C01810=1212.912,107.053,-49.363,-178.523,5.760,148.578
C01811=1212.916,106.785,-49.342,-178.526,5.760,148.579
C01812=1212.922,106.536,-49.323,-178.528,5.758,148.579
C01813=1212.926,106.286,-49.305,-178.531,5.757,148.580
C01814=1212.931,106.037,-49.285,-178.533,5.756,148.581
C01815=1212.935,105.788,-49.266,-178.536,5.755,148.581
C01816=1212.941,105.539,-49.248,-178.539,5.754,148.582
C01817=1212.945,105.289,-49.229,-178.541,5.753,148.582
C01818=1212.950,105.040,-49.209,-178.544,5.752,148.583
C01819=1212.955,104.791,-49.191,-178.546,5.751,148.583
C01820=1212.960,104.542,-49.172,-178.549,5.750,148.584
C01821=1212.965,104.292,-49.154,-178.551,5.749,148.584
C01822=1212.969,104.043,-49.134,-178.554,5.748,148.585
C01823=1212.974,103.794,-49.115,-178.557,5.747,148.585
C01824=1212.979,103.544,-49.097,-178.559,5.746,148.586
C01825=1212.984,103.296,-49.078,-178.562,5.745,148.587
C01826=1212.989,103.046,-49.060,-178.564,5.744,148.587
C01827=1212.993,102.797,-49.040,-178.567,5.743,148.588
C01828=1212.998,102.548,-49.022,-178.570,5.742,148.588
C01829=1213.004,102.299,-49.003,-178.572,5.741,148.589
C01830=1213.008,102.049,-48.985,-178.574,5.740,148.589
C01831=1213.013,101.800,-48.965,-178.578,5.739,148.590
C01832=1213.018,101.550,-48.947,-178.580,5.738,148.590
C01833=1213.022,101.302,-48.928,-178.582,5.737,148.591
C01834=1213.028,101.052,-48.910,-178.585,5.737,148.592
C01835=1213.032,100.803,-48.891,-178.588,5.735,148.592
C01836=1213.037,100.554,-48.873,-178.590,5.734,148.593
C01837=1213.042,100.305,-48.853,-178.593,5.734,148.593
C01838=1213.046,100.055,-48.835,-178.596,5.732,148.594
C01839=1213.052,99.806,-48.816,-178.598,5.731,148.594
C01840=1213.057,99.557,-48.798,-178.600,5.730,148.595
C01841=1213.061,99.308,-48.779,-178.603,5.730,148.595
C01842=1213.066,99.058,-48.760,-178.606,5.728,148.596
C01843=1213.071,98.809,-48.742,-178.608,5.727,148.596
C01844=1213.075,98.560,-48.723,-178.611,5.727,148.597
C01845=1213.081,98.310,-48.704,-178.614,5.725,148.597
C01846=1213.086,98.061,-48.686,-178.616,5.724,148.598
C01847=1213.090,97.812,-48.667,-178.618,5.723,148.599
C01848=1213.095,97.563,-48.649,-178.621,5.723,148.599
C01849=1213.100,97.314,-48.630,-178.624,5.721,148.600
C01850=1213.104,97.064,-48.612,-178.626,5.721,148.600
C01851=1213.109,96.815,-48.594,-178.629,5.720,148.601
C01852=1213.115,96.565,-48.575,-178.632,5.719,148.602
C01853=1213.119,96.316,-48.556,-178.634,5.718,148.602
C01854=1213.124,96.067,-48.538,-178.637,5.717,148.603
C01855=1213.129,95.818,-48.520,-178.639,5.716,148.603
C01856=1213.134,95.569,-48.501,-178.642,5.715,148.604
C01857=1213.138,95.319,-48.483,-178.645,5.714,148.604
C01858=1213.143,95.070,-48.465,-178.647,5.713,148.605
C01859=1213.148,94.821,-48.447,-178.650,5.713,148.605
C01860=1213.154,94.572,-48.427,-178.652,5.711,148.606
C01861=1213.158,94.322,-48.409,-178.655,5.710,148.606
C01862=1213.163,94.073,-48.391,-178.658,5.710,148.607
C01863=1213.168,93.823,-48.373,-178.660,5.709,148.608
C01864=1213.172,93.575,-48.354,-178.663,5.707,148.608
C01865=1213.177,93.325,-48.335,-178.665,5.707,148.609
C01866=1213.182,93.076,-48.317,-178.668,5.706,148.609
C01867=1213.187,92.826,-48.299,-178.670,5.705,148.610
C01868=1213.192,92.577,-48.281,-178.673,5.703,148.610
C01869=1213.196,92.327,-48.263,-178.676,5.703,148.611
C01870=1213.201,92.079,-48.244,-178.678,5.702,148.612
C01871=1213.207,91.829,-48.226,-178.680,5.701,148.612
C01872=1213.212,91.580,-48.208,-178.683,5.700,148.613
C01873=1213.217,91.331,-48.190,-178.686,5.699,148.613
C01874=1213.221,91.081,-48.172,-178.688,5.698,148.614
C01875=1213.226,90.832,-48.154,-178.691,5.698,148.614
C01876=1213.231,90.583,-48.136,-178.694,5.696,148.615
C01877=1213.236,90.334,-48.118,-178.696,5.695,148.615
C01878=1213.241,90.084,-48.100,-178.699,5.695,148.616
C01879=1213.245,89.835,-48.080,-178.701,5.694,148.617
C01880=1213.250,89.586,-48.062,-178.704,5.693,148.617
C01881=1213.255,89.336,-48.044,-178.707,5.692,148.618
C01882=1213.260,89.087,-48.026,-178.709,5.691,148.618
C01883=1213.265,88.838,-48.008,-178.711,5.690,148.619
C01884=1213.270,88.589,-47.990,-178.714,5.690,148.620
C01885=1213.274,88.339,-47.972,-178.717,5.688,148.620
C01886=1213.279,88.090,-47.954,-178.719,5.687,148.621
C01887=1213.284,87.841,-47.936,-178.722,5.687,148.621
C01888=1213.289,87.591,-47.918,-178.724,5.686,148.622
C01889=1213.294,87.342,-47.900,-178.727,5.685,148.622
C01890=1213.299,87.093,-47.882,-178.730,5.684,148.623
C01891=1213.304,86.844,-47.864,-178.732,5.683,148.623
C01892=1213.308,86.594,-47.845,-178.735,5.682,148.624
C01893=1213.313,86.345,-47.828,-178.737,5.681,148.624
C01894=1213.318,86.095,-47.810,-178.740,5.680,148.625
C01895=1213.323,85.846,-47.792,-178.743,5.680,148.626
C01896=1213.328,85.597,-47.774,-178.745,5.679,148.626
C01897=1213.333,85.348,-47.756,-178.747,5.678,148.627
C01898=1213.338,85.098,-47.738,-178.750,5.677,148.628
C01899=1213.343,84.849,-47.720,-178.753,5.676,148.628
C01900=1213.348,84.600,-47.702,-178.755,5.675,148.629
C01901=1213.352,84.350,-47.684,-178.758,5.674,148.629
C01902=1213.357,84.101,-47.666,-178.760,5.674,148.630
C01903=1213.362,83.851,-47.649,-178.763,5.673,148.630
C01904=1213.367,83.602,-47.631,-178.766,5.672,148.631
C01905=1213.372,83.353,-47.613,-178.768,5.671,148.631
C01906=1213.377,83.104,-47.595,-178.771,5.670,148.632
C01907=1213.382,82.855,-47.577,-178.773,5.669,148.633
C01908=1213.387,82.605,-47.559,-178.776,5.669,148.633
C01909=1213.392,82.356,-47.542,-178.779,5.667,148.634
C01910=1213.397,82.106,-47.524,-178.781,5.667,148.634
C01911=1213.401,81.858,-47.506,-178.783,5.666,148.635
C01912=1213.406,81.589,-47.487,-178.786,5.665,148.636
C01913=1213.411,81.320,-47.468,-178.789,5.664,148.636
C01914=1213.416,81.052,-47.449,-178.792,5.663,148.637
C01915=1213.421,80.784,-47.429,-178.795,5.663,148.637
C01916=1213.427,80.534,-47.412,-178.798,5.661,148.638
C01917=1213.432,80.285,-47.394,-178.800,5.660,148.639
C01918=1213.436,80.036,-47.376,-178.803,5.660,148.639
C01919=1213.442,79.786,-47.359,-178.805,5.659,148.640
C01920=1213.447,79.537,-47.341,-178.807,5.658,148.640
C01921=1213.451,79.288,-47.323,-178.810,5.658,148.641
C01922=1213.456,79.038,-47.306,-178.813,5.656,148.642
C01923=1213.461,78.789,-47.288,-178.815,5.655,148.642
C01924=1213.466,78.540,-47.270,-178.818,5.655,148.643
C01925=1213.471,78.290,-47.253,-178.820,5.654,148.643
C01926=1213.476,78.041,-47.235,-178.823,5.653,148.644
C01927=1213.480,77.792,-47.218,-178.825,5.653,148.644
C01928=1213.485,77.542,-47.200,-178.828,5.651,148.645
C01929=1213.490,77.293,-47.182,-178.831,5.651,148.646
C01930=1213.495,77.044,-47.164,-178.833,5.650,148.646
C01931=1213.500,76.794,-47.148,-178.836,5.649,148.647
C01932=1213.505,76.545,-47.130,-178.838,5.649,148.647
C01933=1213.510,76.295,-47.112,-178.841,5.648,148.648
C01934=1213.515,76.046,-47.095,-178.844,5.646,148.649
C01935=1213.520,75.796,-47.077,-178.846,5.646,148.649
C01936=1213.524,75.547,-47.060,-178.849,5.645,148.650
C01937=1213.529,75.298,-47.042,-178.851,5.644,148.650
C01938=1213.534,75.048,-47.025,-178.854,5.644,148.651
C01939=1213.539,74.800,-47.008,-178.856,5.643,148.652
C01940=1213.544,74.551,-46.990,-178.859,5.642,148.652
C01941=1213.549,74.301,-46.972,-178.862,5.641,148.653
C01942=1213.554,74.052,-46.955,-178.864,5.640,148.653
C01943=1213.559,73.803,-46.938,-178.867,5.639,148.654
C01944=1213.564,73.553,-46.920,-178.869,5.639,148.654
C01945=1213.569,73.304,-46.902,-178.872,5.638,148.655
C01946=1213.573,73.054,-46.886,-178.874,5.637,148.656
C01947=1213.578,72.804,-46.869,-178.877,5.637,148.656
C01948=1213.583,72.555,-46.851,-178.880,5.635,148.657
C01949=1213.588,72.306,-46.834,-178.882,5.635,148.657
C01950=1213.593,72.057,-46.816,-178.885,5.634,148.658
C01951=1213.598,71.808,-46.799,-178.887,5.633,148.659
C01952=1213.603,71.559,-46.782,-178.890,5.633,148.659
C01953=1213.608,71.309,-46.764,-178.892,5.632,148.660
C01954=1213.613,71.059,-46.747,-178.895,5.631,148.660
C01955=1213.617,70.810,-46.730,-178.897,5.630,148.661
C01956=1213.622,70.560,-46.712,-178.900,5.629,148.662
C01957=1213.627,70.312,-46.695,-178.903,5.628,148.662
C01958=1213.632,70.062,-46.678,-178.905,5.628,148.663
C01959=1213.638,69.813,-46.661,-178.908,5.627,148.663
C01960=1213.642,69.564,-46.643,-178.910,5.626,148.664
C01961=1213.647,69.314,-46.626,-178.913,5.625,148.664
C01962=1213.652,69.065,-46.610,-178.915,5.625,148.665
C01963=1213.656,68.815,-46.592,-178.918,5.624,148.666
C01964=1213.662,68.566,-46.574,-178.921,5.623,148.666
C01965=1213.666,68.316,-46.558,-178.923,5.622,148.667
C01966=1213.672,68.067,-46.541,-178.926,5.621,148.668
C01967=1213.676,67.818,-46.523,-178.928,5.621,148.668
C01968=1213.681,67.568,-46.506,-178.931,5.620,148.669
C01969=1213.686,67.319,-46.489,-178.933,5.619,148.669
C01970=1213.691,67.070,-46.471,-178.936,5.619,148.670
C01971=1213.696,66.821,-46.455,-178.938,5.618,148.671
C01972=1213.701,66.571,-46.438,-178.941,5.617,148.671
C01973=1213.706,66.322,-46.421,-178.944,5.616,148.672
C01974=1213.711,66.072,-46.404,-178.946,5.615,148.672
C01975=1213.715,65.823,-46.387,-178.949,5.615,148.673
C01976=1213.720,65.573,-46.369,-178.951,5.614,148.673
C01977=1213.725,65.324,-46.353,-178.954,5.613,148.674
C01978=1213.730,65.075,-46.336,-178.956,5.613,148.675
C01979=1213.735,64.825,-46.319,-178.959,5.612,148.675
C01980=1213.740,64.576,-46.301,-178.961,5.611,148.676
C01981=1213.745,64.327,-46.285,-178.964,5.611,148.677
C01982=1213.750,64.077,-46.268,-178.966,5.610,148.677
C01983=1213.755,63.828,-46.251,-178.970,5.609,148.678
C01984=1213.760,63.578,-46.234,-178.972,5.608,148.678
C01985=1213.764,63.329,-46.217,-178.974,5.607,148.679
C01986=1213.770,63.079,-46.200,-178.977,5.607,148.680
C01987=1213.774,62.831,-46.183,-178.980,5.606,148.680
C01988=1213.779,62.581,-46.166,-178.982,5.605,148.681
C01989=1213.785,62.332,-46.149,-178.985,5.605,148.681
C01990=1213.789,62.083,-46.132,-178.987,5.604,148.682
C01991=1213.794,61.833,-46.115,-178.990,5.604,148.683
C01992=1213.799,61.583,-46.098,-178.992,5.603,148.683
C01993=1213.804,61.334,-46.082,-178.995,5.602,148.684
C01994=1213.809,61.085,-46.065,-178.997,5.602,148.685
C01995=1213.814,60.835,-46.048,-179.000,5.600,148.685
C01996=1213.819,60.585,-46.031,-179.003,5.599,148.686
C01997=1213.824,60.337,-46.015,-179.005,5.599,148.686
C01998=1213.828,60.087,-45.998,-179.008,5.598,148.687
C01999=1213.834,59.837,-45.981,-179.010,5.598,148.688
C02000=1213.839,59.589,-45.964,-179.013,5.597,148.688
C02001=1213.843,59.339,-45.948,-179.015,5.596,148.689
C02002=1213.848,59.089,-45.930,-179.018,5.596,148.689
C02003=1213.853,58.840,-45.914,-179.020,5.595,148.690
C02004=1213.858,58.591,-45.898,-179.023,5.594,148.691
C02005=1213.863,58.341,-45.880,-179.025,5.594,148.691
C02006=1213.868,58.092,-45.864,-179.028,5.593,148.692
C02007=1213.873,57.843,-45.847,-179.031,5.592,148.692
C02008=1213.878,57.593,-45.830,-179.033,5.592,148.693
C02009=1213.882,57.344,-45.813,-179.035,5.591,148.694
C02010=1213.887,57.095,-45.797,-179.039,5.590,148.694
C02011=1213.893,56.844,-45.780,-179.041,5.589,148.695
C02012=1213.898,56.596,-45.764,-179.044,5.588,148.696
C02013=1213.903,56.346,-45.748,-179.046,5.588,148.696
C02014=1213.907,56.097,-45.731,-179.049,5.587,148.697
C02015=1213.913,55.848,-45.714,-179.051,5.586,148.697
C02016=1213.918,55.579,-45.696,-179.054,5.586,148.698
C02017=1213.923,55.311,-45.679,-179.056,5.585,148.699
C02018=1213.928,55.042,-45.660,-179.059,5.585,148.699
C02019=1213.934,54.774,-45.642,-179.062,5.583,148.700
C02020=1213.938,54.524,-45.626,-179.065,5.583,148.701
C02021=1213.944,54.275,-45.610,-179.068,5.582,148.701
C02022=1213.949,54.025,-45.593,-179.070,5.581,148.702
C02023=1213.953,53.776,-45.576,-179.072,5.581,148.702
C02024=1213.958,53.527,-45.560,-179.075,5.580,148.703
C02025=1213.963,53.277,-45.544,-179.078,5.580,148.704
C02026=1213.968,53.028,-45.528,-179.080,5.579,148.704
C02027=1213.973,52.778,-45.510,-179.082,5.578,148.705
C02028=1213.978,52.529,-45.494,-179.085,5.578,148.706
C02029=1213.983,52.279,-45.478,-179.088,5.577,148.706
C02030=1213.988,52.030,-45.461,-179.090,5.577,148.707
C02031=1213.993,51.781,-45.445,-179.092,5.576,148.707
C02032=1213.997,51.532,-45.428,-179.095,5.575,148.708
C02033=1214.003,51.282,-45.412,-179.098,5.575,148.709
C02034=1214.008,51.032,-45.396,-179.100,5.574,148.709
C02035=1214.012,50.783,-45.379,-179.103,5.573,148.710
C02036=1214.018,50.533,-45.363,-179.105,5.573,148.710
C02037=1214.022,50.284,-45.347,-179.108,5.572,148.711
C02038=1214.027,50.035,-45.330,-179.110,5.571,148.712
C02039=1214.032,49.785,-45.314,-179.113,5.571,148.712
C02040=1214.037,49.536,-45.298,-179.116,5.570,148.713
C02041=1214.042,49.287,-45.281,-179.118,5.569,148.714
C02042=1214.048,49.037,-45.265,-179.120,5.569,148.714
C02043=1214.052,48.788,-45.249,-179.123,5.568,148.715
C02044=1214.057,48.538,-45.233,-179.126,5.568,148.716
C02045=1214.062,48.289,-45.216,-179.128,5.567,148.716
C02046=1214.067,48.039,-45.200,-179.131,5.566,148.717
C02047=1214.072,47.790,-45.184,-179.133,5.566,148.717
C02048=1214.077,47.540,-45.167,-179.136,5.565,148.718
C02049=1214.082,47.291,-45.152,-179.138,5.565,148.719
C02050=1214.086,47.042,-45.135,-179.141,5.564,148.719
C02051=1214.092,46.792,-45.120,-179.144,5.564,148.720
C02052=1214.096,46.543,-45.103,-179.146,5.563,148.720
C02053=1214.101,46.294,-45.087,-179.149,5.562,148.721
C02054=1214.106,46.044,-45.071,-179.151,5.562,148.722
C02055=1214.111,45.795,-45.054,-179.154,5.561,148.723
C02056=1214.116,45.545,-45.038,-179.156,5.560,148.723
C02057=1214.121,45.296,-45.022,-179.159,5.560,148.724
C02058=1214.126,45.046,-45.006,-179.161,5.559,148.724
C02059=1214.131,44.797,-44.990,-179.164,5.558,148.725
C02060=1214.136,44.548,-44.974,-179.167,5.558,148.726
C02061=1214.141,44.298,-44.958,-179.169,5.557,148.726
C02062=1214.146,44.049,-44.942,-179.171,5.556,148.727
C02063=1214.151,43.799,-44.926,-179.174,5.556,148.727
C02064=1214.156,43.550,-44.910,-179.177,5.555,148.728
C02065=1214.161,43.300,-44.894,-179.179,5.555,148.729
C02066=1214.166,43.051,-44.878,-179.182,5.554,148.729
C02067=1214.171,42.801,-44.862,-179.184,5.554,148.730
C02068=1214.176,42.552,-44.845,-179.187,5.553,148.731
C02069=1214.181,42.303,-44.830,-179.189,5.552,148.731
C02070=1214.186,42.053,-44.814,-179.192,5.552,148.732
C02071=1214.191,41.804,-44.797,-179.195,5.551,148.733
C02072=1214.196,41.554,-44.781,-179.197,5.551,148.733
C02073=1214.201,41.304,-44.766,-179.200,5.550,148.734
C02074=1214.206,41.055,-44.749,-179.202,5.549,148.734
C02075=1214.211,40.806,-44.734,-179.205,5.549,148.735
C02076=1214.216,40.557,-44.717,-179.207,5.548,148.736
C02077=1214.220,40.307,-44.702,-179.210,5.548,148.736
C02078=1214.226,40.058,-44.686,-179.213,5.547,148.737
C02079=1214.230,39.807,-44.670,-179.215,5.546,148.738
C02080=1214.235,39.559,-44.654,-179.217,5.546,148.738
C02081=1214.241,39.309,-44.639,-179.220,5.545,148.739
C02082=1214.246,39.059,-44.623,-179.223,5.544,148.740
C02083=1214.251,38.810,-44.606,-179.225,5.544,148.740
C02084=1214.256,38.561,-44.591,-179.228,5.543,148.741
C02085=1214.260,38.311,-44.575,-179.231,5.543,148.742
C02086=1214.266,38.062,-44.560,-179.233,5.542,148.742
C02087=1214.270,37.812,-44.543,-179.235,5.541,148.743
C02088=1214.275,37.563,-44.527,-179.238,5.541,148.743
C02089=1214.281,37.314,-44.512,-179.241,5.540,148.744
C02090=1214.286,37.063,-44.496,-179.243,5.540,148.745
C02091=1214.290,36.815,-44.480,-179.246,5.539,148.745
C02092=1214.295,36.566,-44.465,-179.248,5.538,148.746
C02093=1214.300,36.315,-44.449,-179.251,5.538,148.746
C02094=1214.306,36.066,-44.433,-179.253,5.537,148.747
C02095=1214.311,35.817,-44.417,-179.256,5.537,148.748
C02096=1214.315,35.567,-44.401,-179.258,5.537,148.749
C02097=1214.320,35.318,-44.386,-179.261,5.536,148.749
C02098=1214.325,35.069,-44.370,-179.263,5.536,148.750
C02099=1214.330,34.819,-44.354,-179.265,5.535,148.750
C02100=1214.335,34.569,-44.339,-179.268,5.534,148.751
C02101=1214.340,34.320,-44.324,-179.271,5.534,148.752
C02102=1214.346,34.071,-44.308,-179.273,5.533,148.752
C02103=1214.350,33.821,-44.291,-179.276,5.533,148.753
C02104=1214.355,33.572,-44.276,-179.279,5.532,148.754
C02105=1214.360,33.323,-44.261,-179.281,5.531,148.754
C02106=1214.365,33.073,-44.245,-179.283,5.531,148.755
C02107=1214.370,32.823,-44.229,-179.286,5.530,148.755
C02108=1214.375,32.574,-44.214,-179.289,5.530,148.756
C02109=1214.380,32.324,-44.198,-179.291,5.529,148.757
C02110=1214.385,32.075,-44.183,-179.294,5.529,148.758
C02111=1214.390,31.825,-44.168,-179.297,5.528,148.758
C02112=1214.395,31.576,-44.152,-179.299,5.527,148.759
C02113=1214.400,31.326,-44.136,-179.301,5.528,148.759
C02114=1214.405,31.077,-44.121,-179.304,5.527,148.760
C02115=1214.410,30.827,-44.106,-179.306,5.527,148.761
C02116=1214.415,30.578,-44.090,-179.309,5.526,148.761
C02117=1214.419,30.328,-44.075,-179.312,5.525,148.762
C02118=1214.425,30.079,-44.059,-179.314,5.525,148.763
C02119=1214.430,29.829,-44.044,-179.316,5.524,148.763
C02120=1214.435,29.561,-44.027,-179.319,5.523,148.764
C02121=1214.441,29.293,-44.010,-179.322,5.523,148.765
C02122=1214.446,29.024,-43.994,-179.325,5.523,148.765
C02123=1214.451,28.755,-43.977,-179.327,5.522,148.766
C02124=1214.456,28.505,-43.961,-179.330,5.522,148.767
C02125=1214.461,28.256,-43.946,-179.332,5.521,148.767
C02126=1214.466,28.007,-43.931,-179.335,5.520,148.768
C02127=1214.471,27.758,-43.915,-179.337,5.520,148.769
C02128=1214.477,27.507,-43.900,-179.340,5.519,148.769
C02129=1214.481,27.258,-43.885,-179.343,5.519,148.770
C02130=1214.487,27.008,-43.869,-179.345,5.518,148.771
C02131=1214.491,26.759,-43.854,-179.348,5.518,148.771
C02132=1214.497,26.510,-43.839,-179.350,5.517,148.772
C02133=1214.501,26.260,-43.824,-179.352,5.517,148.772
C02134=1214.506,26.011,-43.808,-179.355,5.516,148.773
C02135=1214.511,25.761,-43.792,-179.358,5.516,148.774
C02136=1214.516,25.512,-43.778,-179.360,5.515,148.774
C02137=1214.522,25.262,-43.762,-179.363,5.515,148.775
C02138=1214.526,25.013,-43.747,-179.365,5.514,148.776
C02139=1214.531,24.763,-43.732,-179.368,5.514,148.777
C02140=1214.536,24.514,-43.717,-179.370,5.513,148.777
C02141=1214.541,24.264,-43.701,-179.373,5.512,148.778
C02142=1214.546,24.015,-43.687,-179.376,5.512,148.778
C02143=1214.552,23.765,-43.671,-179.378,5.511,148.779
C02144=1214.556,23.516,-43.656,-179.380,5.512,148.780
C02145=1214.561,23.266,-43.640,-179.383,5.511,148.780
C02146=1214.566,23.016,-43.626,-179.386,5.511,148.781
C02147=1214.571,22.767,-43.610,-179.388,5.510,148.782
C02148=1214.576,22.518,-43.595,-179.390,5.509,148.782
C02149=1214.581,22.269,-43.580,-179.393,5.509,148.783
C02150=1214.586,22.019,-43.565,-179.396,5.508,148.784
C02151=1214.592,21.769,-43.550,-179.398,5.508,148.784
C02152=1214.596,21.520,-43.535,-179.401,5.507,148.785
C02153=1214.601,21.270,-43.519,-179.403,5.507,148.786
C02154=1214.606,21.021,-43.505,-179.406,5.507,148.786
C02155=1214.611,20.771,-43.490,-179.408,5.506,148.787
C02156=1214.616,20.522,-43.474,-179.411,5.506,148.788
C02157=1214.621,20.272,-43.460,-179.413,5.505,148.788
C02158=1214.627,20.023,-43.444,-179.416,5.504,148.789
C02159=1214.631,19.774,-43.429,-179.418,5.504,148.789
C02160=1214.637,19.524,-43.414,-179.421,5.503,148.790
C02161=1214.642,19.275,-43.399,-179.423,5.504,148.791
C02162=1214.646,19.025,-43.385,-179.426,5.503,148.791
C02163=1214.652,18.776,-43.369,-179.428,5.503,148.792
C02164=1214.656,18.527,-43.354,-179.431,5.502,148.793
C02165=1214.661,18.276,-43.340,-179.433,5.501,148.793
C02166=1214.666,18.027,-43.324,-179.436,5.501,148.794
C02167=1214.671,17.778,-43.309,-179.439,5.500,148.795
C02168=1214.677,17.528,-43.294,-179.441,5.500,148.795
C02169=1214.681,17.278,-43.279,-179.443,5.500,148.796
C02170=1214.686,17.029,-43.265,-179.446,5.499,148.797
C02171=1214.692,16.779,-43.249,-179.449,5.499,148.797
C02172=1214.697,16.530,-43.235,-179.451,5.498,148.798
C02173=1214.701,16.281,-43.220,-179.454,5.498,148.799
C02174=1214.707,16.031,-43.205,-179.456,5.497,148.799
C02175=1214.712,15.781,-43.190,-179.459,5.496,148.800
C02176=1214.716,15.532,-43.176,-179.461,5.496,148.801
C02177=1214.722,15.282,-43.160,-179.463,5.496,148.801
C02178=1214.727,15.033,-43.146,-179.466,5.496,148.802
C02179=1214.731,14.784,-43.131,-179.469,5.495,148.803
C02180=1214.737,14.534,-43.116,-179.471,5.494,148.803
C02181=1214.742,14.284,-43.101,-179.474,5.494,148.804
C02182=1214.747,14.035,-43.087,-179.477,5.493,148.805
C02183=1214.751,13.786,-43.072,-179.479,5.493,148.805
C02184=1214.757,13.536,-43.057,-179.481,5.493,148.806
C02185=1214.762,13.287,-43.042,-179.484,5.492,148.807
C02186=1214.767,13.037,-43.028,-179.486,5.492,148.807
C02187=1214.771,12.788,-43.013,-179.489,5.491,148.808
C02188=1214.777,12.538,-42.998,-179.491,5.491,148.809
C02189=1214.782,12.288,-42.984,-179.494,5.490,148.809
C02190=1214.787,12.039,-42.969,-179.496,5.491,148.810
C02191=1214.792,11.789,-42.955,-179.499,5.490,148.811
C02192=1214.797,11.540,-42.939,-179.501,5.490,148.811
C02193=1214.802,11.290,-42.925,-179.504,5.489,148.812
C02194=1214.807,11.040,-42.910,-179.506,5.488,148.812
C02195=1214.812,10.791,-42.895,-179.509,5.488,148.813
C02196=1214.817,10.541,-42.881,-179.512,5.487,148.814
C02197=1214.822,10.292,-42.866,-179.514,5.487,148.814
C02198=1214.827,10.042,-42.851,-179.516,5.487,148.815
C02199=1214.832,9.793,-42.837,-179.519,5.486,148.816
C02200=1214.837,9.543,-42.823,-179.522,5.486,148.817
C02201=1214.842,9.295,-42.808,-179.524,5.485,148.817
C02202=1214.848,9.045,-42.793,-179.527,5.485,148.818
C02203=1214.853,8.795,-42.779,-179.529,5.485,148.819
C02204=1214.857,8.546,-42.764,-179.531,5.484,148.819
C02205=1214.862,8.296,-42.750,-179.534,5.484,148.820
C02206=1214.867,8.046,-42.735,-179.536,5.483,148.820
C02207=1214.872,7.797,-42.721,-179.539,5.483,148.821
C02208=1214.878,7.547,-42.706,-179.542,5.482,148.822
C02209=1214.883,7.298,-42.691,-179.544,5.482,148.822
C02210=1214.887,7.048,-42.677,-179.546,5.482,148.823
C02211=1214.892,6.798,-42.663,-179.549,5.481,148.824
C02212=1214.897,6.549,-42.648,-179.552,5.481,148.825
C02213=1214.903,6.300,-42.634,-179.554,5.480,148.825
C02214=1214.908,6.050,-42.619,-179.557,5.480,148.826
C02215=1214.913,5.801,-42.605,-179.559,5.480,148.826
C02216=1214.917,5.552,-42.590,-179.561,5.479,148.827
C02217=1214.923,5.302,-42.575,-179.564,5.479,148.828
C02218=1214.928,5.052,-42.561,-179.567,5.478,148.828
C02219=1214.933,4.802,-42.547,-179.569,5.478,148.829
C02220=1214.938,4.552,-42.533,-179.571,5.478,148.830
C02221=1214.943,4.303,-42.519,-179.574,5.478,148.831
C02222=1214.948,4.054,-42.504,-179.577,5.477,148.831
C02223=1214.953,3.805,-42.489,-179.579,5.476,148.832
C02224=1214.958,3.535,-42.474,-179.582,5.476,148.833
C02225=1214.963,3.266,-42.459,-179.585,5.475,148.833
C02226=1214.969,2.998,-42.443,-179.587,5.475,148.834
C02227=1214.975,2.728,-42.427,-179.590,5.474,148.835
C02228=1214.980,2.479,-42.413,-179.592,5.475,148.835
C02229=1214.985,2.229,-42.399,-179.595,5.474,148.836
C02230=1214.990,1.979,-42.385,-179.597,5.474,148.837
C02231=1214.995,1.730,-42.371,-179.600,5.473,148.837
C02232=1215.000,1.480,-42.356,-179.603,5.473,148.838
C02233=1215.005,1.231,-42.341,-179.605,5.473,148.839
C02234=1215.010,0.982,-42.327,-179.607,5.472,148.839
C02235=1215.015,0.732,-42.313,-179.610,5.472,148.840
C02236=1215.020,0.482,-42.299,-179.613,5.471,148.841
C02237=1215.025,0.233,-42.285,-179.615,5.471,148.842
C02238=1215.030,-0.017,-42.270,-179.617,5.471,148.842
C02239=1215.035,-0.266,-42.257,-179.620,5.470,148.843
C02240=1215.040,-0.515,-42.243,-179.622,5.470,148.843
C02241=1215.045,-0.765,-42.228,-179.625,5.469,148.844
C02242=1215.050,-1.015,-42.214,-179.627,5.469,148.845
C02243=1215.055,-1.264,-42.200,-179.630,5.469,148.845
C02244=1215.060,-1.513,-42.186,-179.632,5.469,148.846
C02245=1215.065,-1.763,-42.172,-179.635,5.468,148.847
C02246=1215.070,-2.013,-42.157,-179.638,5.468,148.847
C02247=1215.075,-2.263,-42.143,-179.640,5.467,148.848
C02248=1215.081,-2.512,-42.129,-179.642,5.467,148.849
C02249=1215.086,-2.762,-42.116,-179.645,5.467,148.850
C02250=1215.091,-3.012,-42.101,-179.648,5.466,148.850
C02251=1215.096,-3.261,-42.087,-179.650,5.466,148.851
C02252=1215.101,-3.510,-42.073,-179.652,5.465,148.851
C02253=1215.106,-3.760,-42.060,-179.654,5.465,148.852
C02254=1215.111,-4.010,-42.045,-179.657,5.465,148.853
C02255=1215.116,-4.259,-42.031,-179.660,5.464,148.853
C02256=1215.121,-4.508,-42.017,-179.662,5.464,148.854
C02257=1215.126,-4.758,-42.003,-179.664,5.464,148.855
C02258=1215.131,-5.008,-41.989,-179.667,5.464,148.856
C02259=1215.137,-5.257,-41.975,-179.670,5.463,148.856
C02260=1215.141,-5.507,-41.962,-179.672,5.463,148.857
C02261=1215.146,-5.756,-41.947,-179.675,5.462,148.858
C02262=1215.151,-6.006,-41.933,-179.677,5.462,148.858
C02263=1215.157,-6.255,-41.919,-179.680,5.462,148.859
C02264=1215.162,-6.505,-41.905,-179.682,5.461,148.860
C02265=1215.167,-6.755,-41.891,-179.685,5.461,148.860
C02266=1215.172,-7.004,-41.878,-179.687,5.461,148.861
C02267=1215.177,-7.254,-41.864,-179.689,5.460,148.862
C02268=1215.182,-7.503,-41.849,-179.692,5.460,148.862
C02269=1215.187,-7.752,-41.836,-179.695,5.459,148.863
C02270=1215.192,-8.003,-41.822,-179.697,5.460,148.864
C02271=1215.197,-8.252,-41.808,-179.699,5.459,148.864
C02272=1215.202,-8.501,-41.794,-179.702,5.459,148.865
C02273=1215.207,-8.751,-41.780,-179.705,5.458,148.866
C02274=1215.212,-9.001,-41.767,-179.707,5.458,148.866
C02275=1215.217,-9.250,-41.753,-179.709,5.458,148.867
C02276=1215.222,-9.499,-41.739,-179.712,5.457,148.868
C02277=1215.227,-9.750,-41.725,-179.715,5.457,148.868
C02278=1215.233,-9.999,-41.711,-179.717,5.456,148.869
C02279=1215.237,-10.248,-41.698,-179.720,5.457,148.870
C02280=1215.242,-10.498,-41.684,-179.722,5.456,148.870
C02281=1215.248,-10.748,-41.670,-179.724,5.455,148.871
C02282=1215.253,-10.997,-41.656,-179.727,5.455,148.872
C02283=1215.257,-11.247,-41.642,-179.729,5.455,148.872
C02284=1215.263,-11.496,-41.629,-179.732,5.455,148.873
C02285=1215.268,-11.746,-41.615,-179.734,5.454,148.874
C02286=1215.272,-11.995,-41.601,-179.737,5.454,148.874
C02287=1215.278,-12.245,-41.588,-179.739,5.454,148.875
C02288=1215.283,-12.495,-41.574,-179.742,5.453,148.876
C02289=1215.289,-12.744,-41.561,-179.744,5.453,148.877
C02290=1215.293,-12.994,-41.547,-179.747,5.452,148.877
C02291=1215.298,-13.243,-41.533,-179.749,5.453,148.878
C02292=1215.304,-13.493,-41.519,-179.752,5.452,148.879
C02293=1215.308,-13.742,-41.506,-179.754,5.452,148.879
C02294=1215.314,-13.992,-41.493,-179.757,5.451,148.880
C02295=1215.319,-14.242,-41.478,-179.759,5.451,148.880
C02296=1215.323,-14.491,-41.465,-179.761,5.451,148.881
C02297=1215.329,-14.741,-41.451,-179.764,5.450,148.882
C02298=1215.333,-14.990,-41.438,-179.767,5.450,148.883
C02299=1215.339,-15.240,-41.424,-179.769,5.450,148.883
C02300=1215.344,-15.490,-41.410,-179.771,5.450,148.884
C02301=1215.349,-15.739,-41.398,-179.774,5.449,148.885
C02302=1215.354,-15.989,-41.383,-179.776,5.449,148.885
C02303=1215.359,-16.239,-41.370,-179.779,5.449,148.886
C02304=1215.364,-16.488,-41.356,-179.781,5.448,148.887
C02305=1215.369,-16.738,-41.343,-179.784,5.448,148.887
C02306=1215.374,-16.987,-41.330,-179.786,5.448,148.888
C02307=1215.380,-17.237,-41.316,-179.789,5.448,148.889
C02308=1215.385,-17.486,-41.302,-179.792,5.447,148.889
C02309=1215.390,-17.736,-41.289,-179.794,5.447,148.890
C02310=1215.395,-17.985,-41.275,-179.796,5.447,148.891
C02311=1215.400,-18.235,-41.262,-179.798,5.446,148.891
C02312=1215.405,-18.484,-41.248,-179.801,5.446,148.892
C02313=1215.410,-18.734,-41.235,-179.804,5.445,148.893
C02314=1215.415,-18.983,-41.221,-179.806,5.446,148.893
C02315=1215.421,-19.233,-41.208,-179.808,5.445,148.894
C02316=1215.426,-19.483,-41.195,-179.811,5.445,148.895
C02317=1215.431,-19.732,-41.181,-179.813,5.445,148.895
C02318=1215.436,-19.982,-41.168,-179.816,5.444,148.896
C02319=1215.441,-20.231,-41.154,-179.819,5.444,148.897
C02320=1215.446,-20.481,-41.142,-179.821,5.443,148.898
C02321=1215.451,-20.731,-41.128,-179.823,5.444,148.898
C02322=1215.456,-20.980,-41.115,-179.826,5.443,148.899
C02323=1215.461,-21.230,-41.101,-179.829,5.443,148.900
C02324=1215.466,-21.479,-41.089,-179.831,5.443,148.900
C02325=1215.471,-21.729,-41.074,-179.833,5.443,148.901
C02326=1215.476,-21.979,-41.062,-179.836,5.442,148.902
C02327=1215.482,-22.229,-41.048,-179.839,5.442,148.902
C02328=1215.486,-22.498,-41.034,-179.841,5.442,148.903
C02329=1215.492,-22.767,-41.019,-179.843,5.441,148.904
C02330=1215.498,-23.037,-41.005,-179.846,5.441,148.905
C02331=1215.503,-23.306,-40.990,-179.849,5.440,148.905
C02332=1215.509,-23.555,-40.977,-179.851,5.440,148.906
C02333=1215.513,-23.805,-40.964,-179.853,5.440,148.907
C02334=1215.519,-24.055,-40.951,-179.856,5.440,148.907
C02335=1215.523,-24.304,-40.937,-179.859,5.439,148.908
C02336=1215.529,-24.554,-40.924,-179.861,5.440,148.909
C02337=1215.534,-24.803,-40.912,-179.864,5.439,148.909
C02338=1215.539,-25.053,-40.899,-179.866,5.439,148.910
C02339=1215.544,-25.302,-40.885,-179.869,5.438,148.911
C02340=1215.549,-25.552,-40.872,-179.871,5.438,148.911
C02341=1215.555,-25.802,-40.858,-179.874,5.438,148.912
C02342=1215.559,-26.052,-40.846,-179.876,5.437,148.913
C02343=1215.564,-26.301,-40.832,-179.878,5.438,148.914
C02344=1215.570,-26.550,-40.819,-179.880,5.437,148.914
C02345=1215.574,-26.800,-40.806,-179.883,5.436,148.915
C02346=1215.580,-27.050,-40.793,-179.885,5.437,148.915
C02347=1215.585,-27.300,-40.780,-179.888,5.436,148.916
C02348=1215.590,-27.549,-40.767,-179.891,5.436,148.917
C02349=1215.596,-27.798,-40.753,-179.893,5.435,148.918
C02350=1215.600,-28.048,-40.740,-179.895,5.436,148.918
C02351=1215.605,-28.298,-40.728,-179.898,5.435,148.919
C02352=1215.610,-28.548,-40.714,-179.901,5.435,148.920
C02353=1215.616,-28.797,-40.702,-179.903,5.435,148.920
C02354=1215.621,-29.047,-40.689,-179.905,5.434,148.921
C02355=1215.626,-29.297,-40.675,-179.908,5.434,148.922
C02356=1215.631,-29.546,-40.662,-179.910,5.434,148.922
C02357=1215.636,-29.795,-40.650,-179.913,5.434,148.923
C02358=1215.641,-30.045,-40.636,-179.915,5.433,148.924
C02359=1215.646,-30.295,-40.623,-179.918,5.434,148.925
C02360=1215.651,-30.545,-40.610,-179.920,5.433,148.925
C02361=1215.657,-30.794,-40.597,-179.923,5.433,148.926
C02362=1215.662,-31.044,-40.585,-179.924,5.433,148.926
C02363=1215.666,-31.294,-40.572,-179.927,5.432,148.927
C02364=1215.671,-31.543,-40.559,-179.930,5.432,148.928
C02365=1215.677,-31.793,-40.546,-179.932,5.431,148.928
C02366=1215.682,-32.043,-40.533,-179.934,5.432,148.929
C02367=1215.687,-32.292,-40.520,-179.937,5.431,148.930
C02368=1215.692,-32.541,-40.508,-179.940,5.431,148.931
C02369=1215.697,-32.792,-40.494,-179.942,5.431,148.931
C02370=1215.702,-33.041,-40.482,-179.945,5.430,148.932
C02371=1215.708,-33.290,-40.469,-179.947,5.430,148.933
C02372=1215.712,-33.540,-40.456,-179.949,5.430,148.933
C02373=1215.718,-33.790,-40.443,-179.952,5.430,148.934
C02374=1215.723,-34.039,-40.430,-179.955,5.429,148.935
C02375=1215.728,-34.289,-40.418,-179.957,5.430,148.935
C02376=1215.733,-34.539,-40.405,-179.959,5.429,148.936
C02377=1215.739,-34.788,-40.391,-179.962,5.429,148.937
C02378=1215.744,-35.038,-40.379,-179.964,5.429,148.938
C02379=1215.748,-35.288,-40.366,-179.967,5.429,148.938
C02380=1215.753,-35.537,-40.353,-179.969,5.428,148.939
C02381=1215.759,-35.786,-40.341,-179.971,5.428,148.939
C02382=1215.764,-36.036,-40.327,-179.974,5.427,148.940
C02383=1215.769,-36.286,-40.314,-179.976,5.427,148.941
C02384=1215.774,-36.535,-40.302,-179.978,5.427,148.942
C02385=1215.779,-36.784,-40.289,-179.981,5.427,148.942
C02386=1215.784,-37.035,-40.277,-179.984,5.426,148.943
C02387=1215.790,-37.285,-40.264,-179.986,5.427,148.944
C02388=1215.795,-37.534,-40.251,-179.988,5.426,148.944
C02389=1215.800,-37.783,-40.239,-179.991,5.426,148.945
C02390=1215.805,-38.033,-40.226,-179.993,5.426,148.946
C02391=1215.810,-38.283,-40.213,-179.996,5.426,148.946
C02392=1215.815,-38.532,-40.200,-179.999,5.425,148.947
C02393=1215.820,-38.782,-40.189,179.999,5.425,148.948
C02394=1215.826,-39.032,-40.175,179.997,5.425,148.949
C02395=1215.831,-39.282,-40.162,179.994,5.425,148.949
C02396=1215.836,-39.531,-40.150,179.992,5.425,148.950
C02397=1215.841,-39.780,-40.137,179.989,5.424,148.951
C02398=1215.846,-40.030,-40.125,179.988,5.424,148.951
C02399=1215.851,-40.280,-40.112,179.985,5.424,148.952
C02400=1215.856,-40.530,-40.100,179.982,5.423,148.952
C02401=1215.861,-40.779,-40.087,179.980,5.424,148.953
C02402=1215.866,-41.028,-40.075,179.978,5.423,148.954
C02403=1215.872,-41.278,-40.063,179.975,5.423,148.955
C02404=1215.876,-41.528,-40.050,179.973,5.423,148.955
C02405=1215.882,-41.778,-40.037,179.970,5.423,148.956
C02406=1215.887,-42.027,-40.024,179.968,5.422,148.957
C02407=1215.893,-42.277,-40.012,179.965,5.422,148.957
C02408=1215.898,-42.526,-39.999,179.963,5.422,148.958
C02409=1215.902,-42.776,-39.986,179.960,5.422,148.959
C02410=1215.907,-43.026,-39.974,179.958,5.422,148.960
C02411=1215.913,-43.276,-39.962,179.955,5.421,148.960
C02412=1215.918,-43.525,-39.949,179.953,5.421,148.961
C02413=1215.923,-43.774,-39.937,179.951,5.421,148.962
C02414=1215.928,-44.025,-39.925,179.948,5.421,148.962
C02415=1215.933,-44.274,-39.912,179.946,5.421,148.963
C02416=1215.938,-44.523,-39.899,179.944,5.420,148.963
C02417=1215.944,-44.773,-39.887,179.941,5.420,148.964
C02418=1215.949,-45.023,-39.875,179.939,5.420,148.965
C02419=1215.954,-45.272,-39.862,179.936,5.420,148.966
C02420=1215.959,-45.522,-39.850,179.934,5.419,148.966
C02421=1215.964,-45.772,-39.837,179.932,5.420,148.967
C02422=1215.969,-46.021,-39.825,179.929,5.419,148.968
C02423=1215.974,-46.271,-39.813,179.926,5.419,148.968
C02424=1215.979,-46.521,-39.800,179.924,5.419,148.969
C02425=1215.985,-46.771,-39.788,179.921,5.418,148.970
C02426=1215.990,-47.020,-39.776,179.919,5.419,148.971
C02427=1215.995,-47.269,-39.763,179.917,5.418,148.971
C02428=1216.001,-47.519,-39.751,179.914,5.418,148.972
C02429=1216.005,-47.769,-39.738,179.912,5.418,148.973
C02430=1216.010,-48.019,-39.727,179.909,5.418,148.973
C02431=1216.015,-48.268,-39.714,179.907,5.417,148.974
C02432=1216.022,-48.538,-39.701,179.905,5.418,148.975
C02433=1216.027,-48.808,-39.688,179.902,5.417,148.975
C02434=1216.032,-49.078,-39.675,179.899,5.417,148.976
C02435=1216.038,-49.348,-39.662,179.897,5.416,148.977
C02436=1216.043,-49.597,-39.649,179.894,5.416,148.978
C02437=1216.048,-49.848,-39.637,179.892,5.416,148.978
C02438=1216.053,-50.097,-39.625,179.890,5.416,148.979
C02439=1216.058,-50.347,-39.613,179.887,5.416,148.980
C02440=1216.063,-50.596,-39.600,179.884,5.415,148.980
C02441=1216.069,-50.846,-39.588,179.882,5.416,148.981
C02442=1216.073,-51.095,-39.576,179.880,5.415,148.982
C02443=1216.079,-51.345,-39.564,179.877,5.415,148.982
C02444=1216.084,-51.594,-39.552,179.875,5.415,148.983
C02445=1216.089,-51.844,-39.540,179.872,5.415,148.984
C02446=1216.094,-52.094,-39.527,179.870,5.415,148.985
C02447=1216.100,-52.344,-39.515,179.868,5.414,148.985
C02448=1216.105,-52.593,-39.503,179.865,5.414,148.986
C02449=1216.110,-52.843,-39.491,179.863,5.414,148.986
C02450=1216.115,-53.093,-39.480,179.861,5.414,148.987
C02451=1216.120,-53.342,-39.467,179.858,5.414,148.988
C02452=1216.126,-53.592,-39.455,179.856,5.413,148.989
C02453=1216.131,-53.841,-39.442,179.853,5.413,148.989
C02454=1216.135,-54.091,-39.431,179.851,5.413,148.990
C02455=1216.140,-54.341,-39.419,179.848,5.413,148.991
C02456=1216.145,-54.591,-39.406,179.846,5.413,148.991
C02457=1216.151,-54.841,-39.394,179.844,5.413,148.992
C02458=1216.156,-55.090,-39.382,179.841,5.412,148.993
C02459=1216.161,-55.340,-39.371,179.839,5.413,148.993
C02460=1216.166,-55.590,-39.359,179.836,5.412,148.994
C02461=1216.171,-55.839,-39.346,179.834,5.412,148.995
C02462=1216.177,-56.089,-39.334,179.831,5.412,148.996
C02463=1216.181,-56.338,-39.323,179.829,5.411,148.996
C02464=1216.186,-56.588,-39.310,179.827,5.412,148.997
C02465=1216.192,-56.838,-39.298,179.825,5.411,148.997
C02466=1216.197,-57.088,-39.287,179.822,5.411,148.998
C02467=1216.202,-57.337,-39.275,179.820,5.411,148.999
C02468=1216.207,-57.587,-39.263,179.817,5.411,149.000
C02469=1216.212,-57.836,-39.251,179.815,5.411,149.000
C02470=1216.218,-58.086,-39.239,179.812,5.410,149.001
C02471=1216.222,-58.335,-39.227,179.810,5.410,149.002
C02472=1216.228,-58.585,-39.215,179.808,5.410,149.002
C02473=1216.233,-58.835,-39.203,179.805,5.410,149.003
C02474=1216.238,-59.084,-39.192,179.803,5.410,149.004
C02475=1216.244,-59.334,-39.180,179.800,5.410,149.005
C02476=1216.249,-59.583,-39.168,179.798,5.410,149.005
C02477=1216.254,-59.833,-39.156,179.796,5.409,149.006
C02478=1216.259,-60.083,-39.145,179.793,5.409,149.006
C02479=1216.265,-60.333,-39.133,179.791,5.409,149.007
C02480=1216.269,-60.582,-39.121,179.788,5.409,149.008
C02481=1216.274,-60.832,-39.109,179.786,5.409,149.009
C02482=1216.280,-61.082,-39.097,179.784,5.409,149.009
C02483=1216.284,-61.331,-39.086,179.781,5.408,149.010
C02484=1216.290,-61.581,-39.074,179.779,5.408,149.011
C02485=1216.295,-61.831,-39.061,179.776,5.408,149.011
C02486=1216.300,-62.080,-39.050,179.774,5.408,149.012
C02487=1216.305,-62.330,-39.038,179.772,5.408,149.013
C02488=1216.311,-62.580,-39.026,179.769,5.407,149.013
C02489=1216.316,-62.829,-39.015,179.767,5.408,149.014
C02490=1216.321,-63.079,-39.003,179.764,5.407,149.015
C02491=1216.326,-63.329,-38.992,179.763,5.407,149.015
C02492=1216.331,-63.578,-38.979,179.760,5.407,149.016
C02493=1216.337,-63.828,-38.967,179.758,5.407,149.017
C02494=1216.341,-64.078,-38.956,179.755,5.407,149.017
C02495=1216.347,-64.328,-38.944,179.752,5.406,149.018
C02496=1216.351,-64.577,-38.933,179.750,5.407,149.019
C02497=1216.357,-64.827,-38.921,179.748,5.406,149.020
C02498=1216.363,-65.076,-38.910,179.746,5.406,149.020
C02499=1216.367,-65.326,-38.898,179.743,5.406,149.021
C02500=1216.373,-65.576,-38.886,179.740,5.406,149.022
C02501=1216.378,-65.826,-38.875,179.738,5.406,149.022
C02502=1216.383,-66.075,-38.863,179.736,5.405,149.023
C02503=1216.388,-66.325,-38.852,179.733,5.406,149.024
C02504=1216.393,-66.575,-38.840,179.731,5.405,149.024
C02505=1216.399,-66.825,-38.828,179.729,5.405,149.025
C02506=1216.404,-67.074,-38.817,179.727,5.405,149.026
C02507=1216.409,-67.324,-38.805,179.724,5.404,149.026
C02508=1216.414,-67.573,-38.794,179.722,5.405,149.027
C02509=1216.419,-67.823,-38.782,179.719,5.404,149.028
C02510=1216.424,-68.073,-38.771,179.717,5.405,149.029
C02511=1216.430,-68.323,-38.759,179.714,5.404,149.029
C02512=1216.435,-68.572,-38.748,179.712,5.405,149.030
C02513=1216.440,-68.822,-38.736,179.710,5.404,149.031
C02514=1216.445,-69.071,-38.725,179.707,5.404,149.031
C02515=1216.450,-69.321,-38.713,179.705,5.404,149.032
C02516=1216.455,-69.571,-38.702,179.703,5.403,149.033
C02517=1216.461,-69.820,-38.690,179.701,5.404,149.033
C02518=1216.466,-70.070,-38.679,179.698,5.403,149.034
C02519=1216.471,-70.320,-38.667,179.696,5.403,149.035
C02520=1216.476,-70.569,-38.656,179.693,5.403,149.035
C02521=1216.481,-70.819,-38.644,179.691,5.403,149.036
C02522=1216.487,-71.068,-38.633,179.688,5.403,149.037
C02523=1216.492,-71.318,-38.621,179.686,5.402,149.038
C02524=1216.497,-71.568,-38.610,179.684,5.403,149.038
C02525=1216.503,-71.818,-38.599,179.681,5.402,149.039
C02526=1216.507,-72.068,-38.587,179.679,5.403,149.040
C02527=1216.512,-72.317,-38.576,179.677,5.402,149.040
C02528=1216.518,-72.567,-38.564,179.675,5.402,149.041
C02529=1216.523,-72.816,-38.553,179.672,5.402,149.042
C02530=1216.528,-73.066,-38.541,179.670,5.402,149.042
C02531=1216.533,-73.315,-38.530,179.667,5.402,149.043
C02532=1216.539,-73.566,-38.519,179.664,5.401,149.044
C02533=1216.544,-73.816,-38.508,179.662,5.402,149.044
C02534=1216.548,-74.065,-38.497,179.660,5.401,149.045
C02535=1216.554,-74.314,-38.485,179.658,5.402,149.046
C02536=1216.560,-74.585,-38.473,179.655,5.401,149.046
C02537=1216.565,-74.856,-38.461,179.652,5.401,149.047
C02538=1216.571,-75.126,-38.449,179.650,5.401,149.048
C02539=1216.576,-75.397,-38.436,179.648,5.401,149.049
C02540=1216.582,-75.647,-38.424,179.645,5.400,149.049
C02541=1216.588,-75.896,-38.414,179.643,5.400,149.050
C02542=1216.592,-76.146,-38.403,179.640,5.400,149.051
C02543=1216.598,-76.396,-38.391,179.638,5.400,149.051
C02544=1216.602,-76.645,-38.380,179.635,5.400,149.052
C02545=1216.608,-76.895,-38.370,179.633,5.400,149.053
C02546=1216.613,-77.145,-38.358,179.631,5.400,149.054
C02547=1216.618,-77.394,-38.346,179.628,5.400,149.054
C02548=1216.623,-77.643,-38.335,179.626,5.399,149.055
C02549=1216.629,-77.894,-38.324,179.624,5.400,149.055
C02550=1216.634,-78.144,-38.313,179.622,5.399,149.056
C02551=1216.639,-78.392,-38.302,179.619,5.399,149.057
C02552=1216.645,-78.643,-38.291,179.617,5.399,149.058
C02553=1216.649,-78.893,-38.280,179.614,5.399,149.058
C02554=1216.654,-79.142,-38.268,179.612,5.399,149.059
C02555=1216.660,-79.392,-38.258,179.609,5.399,149.060
C02556=1216.665,-79.642,-38.246,179.607,5.399,149.060
C02557=1216.670,-79.891,-38.235,179.605,5.398,149.061
C02558=1216.676,-80.141,-38.225,179.603,5.399,149.062
C02559=1216.681,-80.391,-38.213,179.600,5.398,149.062
C02560=1216.686,-80.640,-38.202,179.598,5.398,149.063
C02561=1216.691,-80.890,-38.191,179.596,5.398,149.064
C02562=1216.696,-81.140,-38.180,179.593,5.398,149.064
C02563=1216.702,-81.390,-38.169,179.591,5.398,149.065
C02564=1216.707,-81.639,-38.158,179.588,5.397,149.066
C02565=1216.712,-81.889,-38.147,179.586,5.398,149.067
C02566=1216.717,-82.139,-38.136,179.583,5.397,149.067
C02567=1216.723,-82.388,-38.125,179.582,5.397,149.068
C02568=1216.728,-82.638,-38.114,179.579,5.397,149.068
C02569=1216.733,-82.887,-38.103,179.577,5.397,149.069
C02570=1216.738,-83.137,-38.092,179.574,5.397,149.070
C02571=1216.743,-83.387,-38.081,179.572,5.397,149.071
C02572=1216.749,-83.637,-38.070,179.570,5.397,149.071
C02573=1216.754,-83.887,-38.059,179.568,5.397,149.072
C02574=1216.758,-84.136,-38.048,179.565,5.397,149.073
C02575=1216.764,-84.386,-38.038,179.563,5.397,149.073
C02576=1216.769,-84.636,-38.026,179.561,5.396,149.074
C02577=1216.775,-84.885,-38.016,179.558,5.397,149.075
C02578=1216.780,-85.135,-38.004,179.556,5.396,149.075
C02579=1216.785,-85.385,-37.994,179.553,5.396,149.076
C02580=1216.790,-85.634,-37.983,179.551,5.396,149.077
C02581=1216.795,-85.884,-37.972,179.548,5.396,149.077
C02582=1216.800,-86.133,-37.961,179.546,5.396,149.078
C02583=1216.806,-86.384,-37.950,179.544,5.396,149.079
C02584=1216.811,-86.634,-37.939,179.542,5.396,149.079
C02585=1216.816,-86.883,-37.929,179.539,5.395,149.080
C02586=1216.821,-87.133,-37.917,179.537,5.395,149.081
C02587=1216.827,-87.382,-37.907,179.535,5.395,149.082
C02588=1216.831,-87.632,-37.896,179.532,5.395,149.082
C02589=1216.836,-87.882,-37.885,179.530,5.395,149.083
C02590=1216.842,-88.131,-37.874,179.528,5.395,149.084
C02591=1216.847,-88.382,-37.863,179.525,5.395,149.084
C02592=1216.853,-88.631,-37.853,179.523,5.395,149.085
C02593=1216.858,-88.881,-37.842,179.521,5.394,149.086
C02594=1216.863,-89.130,-37.831,179.519,5.395,149.086
C02595=1216.868,-89.380,-37.820,179.516,5.394,149.087
C02596=1216.873,-89.629,-37.810,179.514,5.395,149.088
C02597=1216.878,-89.880,-37.799,179.511,5.394,149.088
C02598=1216.883,-90.129,-37.788,179.509,5.395,149.089
C02599=1216.889,-90.379,-37.778,179.506,5.394,149.090
C02600=1216.894,-90.629,-37.767,179.505,5.394,149.090
C02601=1216.899,-90.878,-37.756,179.502,5.394,149.091
C02602=1216.904,-91.128,-37.746,179.500,5.394,149.092
C02603=1216.910,-91.378,-37.736,179.497,5.394,149.092
C02604=1216.915,-91.628,-37.724,179.495,5.393,149.093
C02605=1216.921,-91.877,-37.713,179.493,5.394,149.094
C02606=1216.926,-92.128,-37.703,179.490,5.393,149.095
C02607=1216.931,-92.377,-37.692,179.488,5.393,149.095
C02608=1216.936,-92.627,-37.681,179.486,5.393,149.096
C02609=1216.942,-92.876,-37.671,179.484,5.393,149.096
C02610=1216.946,-93.126,-37.660,179.481,5.393,149.097
C02611=1216.952,-93.375,-37.650,179.479,5.393,149.098
C02612=1216.957,-93.626,-37.639,179.476,5.393,149.099
C02613=1216.962,-93.875,-37.629,179.474,5.393,149.099
C02614=1216.967,-94.125,-37.618,179.471,5.393,149.100
C02615=1216.973,-94.374,-37.607,179.470,5.393,149.101
C02616=1216.978,-94.625,-37.597,179.467,5.392,149.101
C02617=1216.983,-94.874,-37.587,179.465,5.392,149.102
C02618=1216.988,-95.124,-37.575,179.462,5.392,149.103
C02619=1216.994,-95.373,-37.565,179.460,5.392,149.103
C02620=1216.999,-95.624,-37.555,179.458,5.392,149.104
C02621=1217.004,-95.873,-37.544,179.456,5.392,149.105
C02622=1217.010,-96.122,-37.533,179.453,5.392,149.105
C02623=1217.015,-96.372,-37.523,179.451,5.392,149.106
C02624=1217.020,-96.622,-37.513,179.449,5.391,149.107
C02625=1217.024,-96.872,-37.503,179.447,5.392,149.107
C02626=1217.030,-97.121,-37.492,179.444,5.391,149.108
C02627=1217.035,-97.371,-37.481,179.442,5.392,149.109
C02628=1217.040,-97.621,-37.471,179.440,5.391,149.109
C02629=1217.045,-97.871,-37.460,179.437,5.391,149.110
C02630=1217.051,-98.120,-37.450,179.435,5.391,149.111
C02631=1217.056,-98.370,-37.440,179.433,5.391,149.111
C02632=1217.061,-98.620,-37.429,179.430,5.391,149.112
C02633=1217.067,-98.870,-37.419,179.428,5.391,149.113
C02634=1217.072,-99.119,-37.408,179.425,5.391,149.114
C02635=1217.077,-99.369,-37.398,179.424,5.391,149.114
C02636=1217.082,-99.619,-37.387,179.421,5.390,149.115
C02637=1217.087,-99.868,-37.377,179.419,5.391,149.116
C02638=1217.093,-100.118,-37.367,179.416,5.390,149.116
C02639=1217.098,-100.368,-37.357,179.414,5.391,149.117
C02640=1217.104,-100.639,-37.346,179.411,5.390,149.118
C02641=1217.110,-100.910,-37.335,179.409,5.391,149.118
C02642=1217.115,-101.182,-37.323,179.407,5.390,149.119
C02643=1217.120,-101.453,-37.311,179.404,5.390,149.120
C02644=1217.126,-101.702,-37.301,179.402,5.390,149.121
C02645=1217.132,-101.952,-37.291,179.399,5.390,149.121
C02646=1217.137,-102.202,-37.280,179.397,5.390,149.122
C02647=1217.141,-102.451,-37.271,179.395,5.389,149.122
C02648=1217.146,-102.701,-37.260,179.393,5.390,149.123
C02649=1217.152,-102.951,-37.250,179.390,5.389,149.124
C02650=1217.158,-103.200,-37.240,179.388,5.390,149.125
C02651=1217.163,-103.451,-37.229,179.385,5.389,149.125
C02652=1217.168,-103.700,-37.219,179.383,5.390,149.126
C02653=1217.173,-103.949,-37.209,179.381,5.389,149.126
C02654=1217.178,-104.200,-37.199,179.379,5.389,149.127
C02655=1217.184,-104.449,-37.189,179.377,5.390,149.128
C02656=1217.189,-104.699,-37.178,179.374,5.389,149.129
C02657=1217.194,-104.949,-37.168,179.372,5.389,149.129
C02658=1217.199,-105.198,-37.158,179.370,5.389,149.130
C02659=1217.205,-105.448,-37.148,179.368,5.389,149.131
C02660=1217.210,-105.698,-37.137,179.365,5.389,149.131
C02661=1217.215,-105.948,-37.127,179.363,5.389,149.132
C02662=1217.220,-106.197,-37.118,179.360,5.389,149.133
C02663=1217.225,-106.447,-37.107,179.358,5.389,149.133
C02664=1217.231,-106.697,-37.098,179.356,5.389,149.134
C02665=1217.237,-106.947,-37.087,179.354,5.389,149.135
C02666=1217.241,-107.197,-37.077,179.351,5.388,149.135
C02667=1217.246,-107.446,-37.067,179.349,5.388,149.136
C02668=1217.252,-107.696,-37.057,179.347,5.388,149.137
C02669=1217.257,-107.946,-37.046,179.345,5.388,149.137
C02670=1217.262,-108.195,-37.037,179.342,5.388,149.138
C02671=1217.268,-108.445,-37.027,179.340,5.388,149.139
C02672=1217.273,-108.695,-37.016,179.338,5.388,149.139
C02673=1217.278,-108.945,-37.007,179.336,5.388,149.140
C02674=1217.283,-109.194,-36.997,179.333,5.388,149.141
C02675=1217.289,-109.444,-36.987,179.331,5.388,149.141
C02676=1217.294,-109.694,-36.976,179.329,5.387,149.142
C02677=1217.299,-109.944,-36.966,179.326,5.387,149.143
C02678=1217.304,-110.193,-36.956,179.324,5.387,149.143
C02679=1217.310,-110.444,-36.946,179.322,5.387,149.144
C02680=1217.315,-110.693,-36.937,179.319,5.387,149.145
C02681=1217.320,-110.943,-36.927,179.317,5.387,149.145
C02682=1217.326,-111.192,-36.916,179.315,5.387,149.146
C02683=1217.330,-111.442,-36.906,179.313,5.387,149.147
C02684=1217.336,-111.692,-36.897,179.311,5.387,149.147
C02685=1217.341,-111.942,-36.887,179.308,5.387,149.148
C02686=1217.346,-112.191,-36.877,179.306,5.387,149.149
C02687=1217.351,-112.441,-36.867,179.304,5.387,149.149
C02688=1217.357,-112.691,-36.856,179.302,5.387,149.150
C02689=1217.362,-112.941,-36.847,179.299,5.386,149.151
C02690=1217.368,-113.190,-36.837,179.297,5.387,149.152
C02691=1217.372,-113.440,-36.827,179.295,5.386,149.152
C02692=1217.378,-113.690,-36.817,179.292,5.386,149.153
C02693=1217.383,-113.940,-36.808,179.290,5.386,149.153
C02694=1217.388,-114.189,-36.798,179.288,5.386,149.154
C02695=1217.394,-114.439,-36.788,179.285,5.386,149.155
C02696=1217.399,-114.690,-36.778,179.283,5.386,149.155
C02697=1217.404,-114.939,-36.768,179.281,5.386,149.156
C02698=1217.410,-115.188,-36.758,179.279,5.386,149.157
C02699=1217.415,-115.438,-36.748,179.277,5.386,149.157
C02700=1217.420,-115.688,-36.739,179.274,5.386,149.158
C02701=1217.425,-115.938,-36.729,179.272,5.386,149.159
C02702=1217.430,-116.187,-36.719,179.270,5.386,149.159
C02703=1217.436,-116.437,-36.709,179.268,5.386,149.160
C02704=1217.441,-116.687,-36.700,179.265,5.385,149.161
C02705=1217.447,-116.936,-36.689,179.263,5.385,149.161
C02706=1217.451,-117.187,-36.680,179.261,5.385,149.162
C02707=1217.457,-117.436,-36.670,179.258,5.385,149.163
C02708=1217.462,-117.686,-36.661,179.256,5.385,149.163
C02709=1217.468,-117.936,-36.651,179.254,5.385,149.164
C02710=1217.472,-118.185,-36.641,179.252,5.385,149.165
C02711=1217.478,-118.435,-36.632,179.249,5.385,149.165
C02712=1217.483,-118.685,-36.622,179.247,5.385,149.166
C02713=1217.488,-118.935,-36.612,179.245,5.385,149.167
C02714=1217.493,-119.184,-36.603,179.243,5.385,149.167
C02715=1217.499,-119.434,-36.592,179.240,5.385,149.168
C02716=1217.504,-119.684,-36.584,179.238,5.385,149.169
C02717=1217.510,-119.933,-36.573,179.236,5.385,149.169
C02718=1217.514,-120.184,-36.564,179.234,5.385,149.170
C02719=1217.520,-120.433,-36.554,179.231,5.384,149.171
C02720=1217.525,-120.683,-36.544,179.229,5.384,149.171
C02721=1217.531,-120.933,-36.535,179.227,5.384,149.172
C02722=1217.536,-121.182,-36.525,179.224,5.384,149.173
C02723=1217.541,-121.432,-36.516,179.222,5.384,149.173
C02724=1217.546,-121.681,-36.506,179.220,5.384,149.174
C02725=1217.552,-121.932,-36.496,179.218,5.384,149.175
C02726=1217.556,-122.182,-36.487,179.215,5.384,149.175
C02727=1217.562,-122.432,-36.477,179.214,5.384,149.176
C02728=1217.567,-122.681,-36.467,179.211,5.384,149.177
C02729=1217.573,-122.931,-36.458,179.209,5.384,149.177
C02730=1217.578,-123.180,-36.448,179.206,5.384,149.178
C02731=1217.583,-123.430,-36.439,179.205,5.384,149.179
C02732=1217.589,-123.680,-36.429,179.202,5.383,149.179
C02733=1217.594,-123.930,-36.420,179.200,5.384,149.180
C02734=1217.599,-124.180,-36.410,179.197,5.383,149.181
C02735=1217.604,-124.430,-36.401,179.196,5.383,149.181
C02736=1217.610,-124.680,-36.391,179.193,5.383,149.182
C02737=1217.615,-124.929,-36.382,179.191,5.383,149.183
C02738=1217.620,-125.179,-36.373,179.189,5.384,149.183
C02739=1217.626,-125.428,-36.363,179.187,5.383,149.184
C02740=1217.631,-125.678,-36.354,179.185,5.383,149.185
C02741=1217.636,-125.928,-36.344,179.182,5.383,149.185
C02742=1217.642,-126.178,-36.335,179.180,5.383,149.186
C02743=1217.647,-126.428,-36.326,179.178,5.382,149.186
C02744=1217.225,-126.438,-36.362,179.173,5.386,149.189
C02745=1217.220,-126.188,-36.371,179.176,5.386,149.188
C02746=1217.214,-125.939,-36.381,179.178,5.386,149.187
C02747=1217.209,-125.689,-36.390,179.180,5.387,149.187
C02748=1217.204,-125.440,-36.400,179.182,5.386,149.186
C02749=1217.198,-125.190,-36.409,179.185,5.387,149.185
C02750=1217.193,-124.940,-36.418,179.187,5.386,149.185
C02751=1217.188,-124.690,-36.429,179.189,5.386,149.184
C02752=1217.183,-124.440,-36.438,179.191,5.387,149.183
C02753=1217.178,-124.190,-36.447,179.193,5.386,149.183
C02754=1217.172,-123.940,-36.457,179.196,5.387,149.182
C02755=1217.167,-123.691,-36.466,179.198,5.387,149.181
C02756=1217.161,-123.441,-36.476,179.200,5.387,149.181
C02757=1217.157,-123.192,-36.485,179.202,5.387,149.180
C02758=1217.151,-122.942,-36.495,179.205,5.387,149.179
C02759=1217.146,-122.692,-36.505,179.207,5.387,149.179
C02760=1217.141,-122.442,-36.513,179.209,5.388,149.178
C02761=1217.136,-122.192,-36.524,179.211,5.387,149.177
C02762=1217.130,-121.942,-36.533,179.214,5.387,149.177
C02763=1217.125,-121.693,-36.543,179.216,5.388,149.176
C02764=1217.120,-121.443,-36.552,179.218,5.387,149.175
C02765=1217.114,-121.193,-36.562,179.221,5.388,149.175
C02766=1217.109,-120.944,-36.571,179.223,5.387,149.174
C02767=1217.103,-120.694,-36.581,179.225,5.388,149.173
C02768=1217.098,-120.444,-36.590,179.227,5.388,149.173
C02769=1217.093,-120.194,-36.601,179.230,5.388,149.172
C02770=1217.088,-119.944,-36.610,179.232,5.388,149.171
C02771=1217.082,-119.695,-36.620,179.234,5.388,149.171
C02772=1217.078,-119.445,-36.629,179.236,5.388,149.170
C02773=1217.072,-119.195,-36.639,179.239,5.389,149.169
C02774=1217.067,-118.946,-36.649,179.241,5.388,149.169
C02775=1217.061,-118.695,-36.658,179.243,5.388,149.168
C02776=1217.057,-118.446,-36.668,179.245,5.389,149.168
C02777=1217.051,-118.196,-36.678,179.247,5.388,149.167
C02778=1217.046,-117.946,-36.687,179.250,5.389,149.166
C02779=1217.040,-117.697,-36.697,179.252,5.388,149.165
C02780=1217.035,-117.447,-36.706,179.254,5.389,149.165
C02781=1217.030,-117.197,-36.717,179.256,5.389,149.164
C02782=1217.025,-116.948,-36.726,179.259,5.389,149.163
C02783=1217.019,-116.697,-36.736,179.261,5.389,149.163
C02784=1217.014,-116.448,-36.746,179.264,5.389,149.162
C02785=1217.009,-116.199,-36.756,179.265,5.389,149.162
C02786=1217.004,-115.948,-36.766,179.268,5.389,149.161
C02787=1216.999,-115.698,-36.775,179.270,5.389,149.160
C02788=1216.993,-115.449,-36.785,179.273,5.389,149.159
C02789=1216.988,-115.199,-36.794,179.274,5.390,149.159
C02790=1216.982,-114.950,-36.805,179.276,5.389,149.158
C02791=1216.978,-114.700,-36.815,179.279,5.390,149.157
C02792=1216.972,-114.449,-36.824,179.281,5.389,149.157
C02793=1216.967,-114.200,-36.834,179.284,5.390,149.156
C02794=1216.962,-113.951,-36.844,179.285,5.390,149.156
C02795=1216.956,-113.701,-36.854,179.288,5.390,149.155
C02796=1216.952,-113.451,-36.863,179.290,5.390,149.154
C02797=1216.946,-113.201,-36.874,179.293,5.390,149.153
C02798=1216.940,-112.951,-36.884,179.295,5.390,149.153
C02799=1216.935,-112.702,-36.893,179.297,5.390,149.152
C02800=1216.930,-112.451,-36.903,179.299,5.390,149.151
C02801=1216.925,-112.202,-36.913,179.302,5.390,149.151
C02802=1216.920,-111.953,-36.923,179.304,5.390,149.150
C02803=1216.914,-111.703,-36.933,179.307,5.391,149.149
C02804=1216.908,-111.453,-36.943,179.308,5.391,149.149
C02805=1216.904,-111.203,-36.953,179.311,5.391,149.148
C02806=1216.898,-110.953,-36.963,179.313,5.391,149.147
C02807=1216.893,-110.704,-36.973,179.315,5.390,149.147
C02808=1216.888,-110.454,-36.983,179.318,5.391,149.146
C02809=1216.883,-110.204,-36.993,179.319,5.391,149.146
C02810=1216.877,-109.954,-37.003,179.322,5.391,149.145
C02811=1216.872,-109.705,-37.012,179.324,5.391,149.144
C02812=1216.867,-109.455,-37.023,179.327,5.391,149.143
C02813=1216.862,-109.205,-37.033,179.329,5.391,149.143
C02814=1216.857,-108.956,-37.043,179.331,5.391,149.142
C02815=1216.851,-108.706,-37.052,179.333,5.391,149.141
C02816=1216.846,-108.456,-37.063,179.336,5.392,149.141
C02817=1216.840,-108.206,-37.073,179.338,5.391,149.140
C02818=1216.835,-107.957,-37.083,179.341,5.392,149.139
C02819=1216.830,-107.707,-37.093,179.342,5.392,149.139
C02820=1216.825,-107.457,-37.104,179.345,5.392,149.138
C02821=1216.820,-107.208,-37.113,179.347,5.392,149.137
C02822=1216.815,-106.958,-37.124,179.350,5.392,149.137
C02823=1216.809,-106.707,-37.133,179.352,5.392,149.136
C02824=1216.803,-106.458,-37.143,179.354,5.392,149.135
C02825=1216.799,-106.208,-37.153,179.356,5.392,149.135
C02826=1216.793,-105.958,-37.164,179.359,5.393,149.134
C02827=1216.788,-105.709,-37.174,179.361,5.392,149.133
C02828=1216.783,-105.459,-37.184,179.363,5.393,149.133
C02829=1216.778,-105.209,-37.194,179.366,5.392,149.132
C02830=1216.772,-104.960,-37.204,179.368,5.393,149.131
C02831=1216.767,-104.710,-37.215,179.370,5.393,149.131
C02832=1216.762,-104.460,-37.225,179.373,5.393,149.130
C02833=1216.756,-104.210,-37.235,179.375,5.393,149.129
C02834=1216.752,-103.961,-37.245,179.377,5.393,149.129
C02835=1216.746,-103.711,-37.255,179.379,5.393,149.128
C02836=1216.741,-103.461,-37.266,179.381,5.393,149.127
C02837=1216.736,-103.211,-37.276,179.384,5.393,149.127
C02838=1216.730,-102.962,-37.286,179.386,5.393,149.126
C02839=1216.725,-102.712,-37.296,179.388,5.393,149.125
C02840=1216.720,-102.462,-37.307,179.391,5.393,149.125
C02841=1216.715,-102.213,-37.317,179.393,5.393,149.124
C02842=1216.710,-101.962,-37.327,179.395,5.393,149.123
C02843=1216.704,-101.713,-37.338,179.397,5.394,149.123
C02844=1216.699,-101.463,-37.348,179.400,5.393,149.122
C02845=1216.693,-101.192,-37.359,179.402,5.394,149.121
C02846=1216.687,-100.920,-37.370,179.405,5.394,149.120
C02847=1216.682,-100.650,-37.382,179.407,5.394,149.120
C02848=1216.677,-100.379,-37.392,179.410,5.394,149.119
C02849=1216.672,-100.129,-37.403,179.412,5.394,149.118
C02850=1216.666,-99.879,-37.413,179.414,5.394,149.118
C02851=1216.661,-99.630,-37.423,179.417,5.394,149.117
C02852=1216.656,-99.380,-37.434,179.419,5.394,149.116
C02853=1216.650,-99.130,-37.444,179.421,5.394,149.115
C02854=1216.645,-98.880,-37.455,179.423,5.395,149.115
C02855=1216.639,-98.630,-37.465,179.426,5.394,149.114
C02856=1216.635,-98.381,-37.476,179.428,5.395,149.114
C02857=1216.630,-98.131,-37.486,179.430,5.394,149.113
C02858=1216.624,-97.882,-37.496,179.433,5.395,149.112
C02859=1216.619,-97.632,-37.507,179.435,5.395,149.111
C02860=1216.614,-97.382,-37.517,179.438,5.395,149.111
C02861=1216.609,-97.132,-37.528,179.439,5.395,149.110
C02862=1216.603,-96.882,-37.538,179.442,5.395,149.110
C02863=1216.598,-96.633,-37.549,179.444,5.395,149.109
C02864=1216.593,-96.383,-37.559,179.447,5.395,149.108
C02865=1216.587,-96.134,-37.569,179.449,5.395,149.107
C02866=1216.582,-95.883,-37.580,179.452,5.395,149.107
C02867=1216.577,-95.634,-37.590,179.453,5.396,149.106
C02868=1216.572,-95.384,-37.601,179.456,5.396,149.105
C02869=1216.566,-95.135,-37.612,179.458,5.396,149.105
C02870=1216.561,-94.884,-37.622,179.461,5.396,149.104
C02871=1216.556,-94.635,-37.632,179.463,5.396,149.103
C02872=1216.551,-94.385,-37.644,179.465,5.396,149.103
C02873=1216.545,-94.136,-37.654,179.467,5.396,149.102
C02874=1216.540,-93.885,-37.665,179.470,5.397,149.101
C02875=1216.535,-93.636,-37.675,179.472,5.396,149.101
C02876=1216.530,-93.386,-37.686,179.474,5.397,149.100
C02877=1216.524,-93.137,-37.696,179.477,5.396,149.099
C02878=1216.519,-92.886,-37.707,179.479,5.397,149.099
C02879=1216.514,-92.637,-37.717,179.482,5.397,149.098
C02880=1216.509,-92.387,-37.728,179.484,5.397,149.097
C02881=1216.504,-92.138,-37.739,179.486,5.398,149.097
C02882=1216.499,-91.887,-37.749,179.488,5.397,149.096
C02883=1216.493,-91.639,-37.760,179.491,5.398,149.095
C02884=1216.488,-91.388,-37.771,179.493,5.397,149.095
C02885=1216.483,-91.139,-37.781,179.496,5.398,149.094
C02886=1216.478,-90.889,-37.792,179.498,5.397,149.093
C02887=1216.472,-90.640,-37.802,179.500,5.398,149.092
C02888=1216.467,-90.389,-37.813,179.502,5.398,149.092
C02889=1216.462,-90.140,-37.824,179.505,5.398,149.091
C02890=1216.457,-89.890,-37.834,179.507,5.398,149.091
C02891=1216.452,-89.641,-37.845,179.509,5.398,149.090
C02892=1216.446,-89.391,-37.856,179.512,5.398,149.089
C02893=1216.441,-89.141,-37.867,179.514,5.398,149.088
C02894=1216.436,-88.892,-37.878,179.516,5.398,149.088
C02895=1216.431,-88.641,-37.889,179.519,5.398,149.087
C02896=1216.425,-88.392,-37.899,179.521,5.398,149.086
C02897=1216.421,-88.142,-37.910,179.523,5.399,149.086
C02898=1216.415,-87.893,-37.920,179.525,5.398,149.085
C02899=1216.410,-87.643,-37.932,179.528,5.399,149.084
C02900=1216.405,-87.393,-37.942,179.530,5.399,149.084
C02901=1216.400,-87.144,-37.953,179.533,5.399,149.083
C02902=1216.394,-86.893,-37.964,179.535,5.399,149.082
C02903=1216.389,-86.644,-37.975,179.538,5.399,149.081
C02904=1216.384,-86.394,-37.986,179.539,5.399,149.081
C02905=1216.378,-86.145,-37.996,179.542,5.400,149.080
C02906=1216.374,-85.895,-38.007,179.545,5.400,149.080
C02907=1216.368,-85.645,-38.017,179.547,5.400,149.079
C02908=1216.363,-85.396,-38.029,179.549,5.400,149.078
C02909=1216.358,-85.145,-38.040,179.551,5.400,149.077
C02910=1216.352,-84.896,-38.051,179.554,5.400,149.077
C02911=1216.347,-84.646,-38.061,179.556,5.400,149.076
C02912=1216.343,-84.396,-38.073,179.558,5.401,149.076
C02913=1216.337,-84.147,-38.083,179.560,5.400,149.075
C02914=1216.332,-83.897,-38.095,179.563,5.401,149.074
C02915=1216.326,-83.648,-38.106,179.565,5.400,149.073
C02916=1216.321,-83.398,-38.116,179.568,5.401,149.073
C02917=1216.317,-83.148,-38.128,179.570,5.400,149.072
C02918=1216.311,-82.899,-38.138,179.573,5.401,149.071
C02919=1216.306,-82.649,-38.150,179.575,5.400,149.071
C02920=1216.301,-82.398,-38.160,179.577,5.401,149.070
C02921=1216.295,-82.149,-38.171,179.579,5.401,149.069
C02922=1216.291,-81.900,-38.182,179.582,5.401,149.069
C02923=1216.285,-81.650,-38.193,179.584,5.402,149.068
C02924=1216.280,-81.400,-38.205,179.586,5.401,149.067
C02925=1216.275,-81.150,-38.215,179.589,5.402,149.067
C02926=1216.269,-80.901,-38.226,179.591,5.401,149.066
C02927=1216.265,-80.652,-38.237,179.594,5.402,149.065
C02928=1216.259,-80.401,-38.249,179.596,5.402,149.064
C02929=1216.254,-80.152,-38.259,179.599,5.402,149.064
C02930=1216.249,-79.902,-38.270,179.600,5.402,149.063
C02931=1216.243,-79.652,-38.282,179.603,5.402,149.063
C02932=1216.238,-79.403,-38.293,179.605,5.402,149.062
C02933=1216.233,-79.153,-38.303,179.608,5.403,149.061
C02934=1216.228,-78.903,-38.315,179.610,5.402,149.060
C02935=1216.222,-78.654,-38.326,179.612,5.403,149.060
C02936=1216.217,-78.404,-38.337,179.615,5.403,149.059
C02937=1216.212,-78.154,-38.348,179.617,5.403,149.058
C02938=1216.207,-77.904,-38.360,179.620,5.403,149.058
C02939=1216.202,-77.655,-38.371,179.621,5.403,149.057
C02940=1216.197,-77.405,-38.381,179.624,5.404,149.056
C02941=1216.191,-77.155,-38.393,179.626,5.403,149.056
C02942=1216.186,-76.906,-38.404,179.629,5.404,149.055
C02943=1216.181,-76.656,-38.415,179.631,5.403,149.054
C02944=1216.176,-76.406,-38.427,179.634,5.404,149.054
C02945=1216.170,-76.157,-38.438,179.636,5.403,149.053
C02946=1216.166,-75.907,-38.449,179.638,5.404,149.052
C02947=1216.160,-75.657,-38.460,179.641,5.404,149.051
C02948=1216.155,-75.407,-38.471,179.643,5.404,149.051
C02949=1216.149,-75.137,-38.483,179.646,5.404,149.050
C02950=1216.144,-74.866,-38.496,179.648,5.405,149.049
C02951=1216.138,-74.595,-38.508,179.651,5.405,149.049
C02952=1216.133,-74.326,-38.520,179.653,5.405,149.048
C02953=1216.127,-74.076,-38.532,179.655,5.405,149.047
C02954=1216.122,-73.826,-38.543,179.658,5.405,149.046
C02955=1216.116,-73.577,-38.554,179.661,5.406,149.046
C02956=1216.111,-73.326,-38.565,179.663,5.405,149.045
C02957=1216.107,-73.077,-38.576,179.665,5.406,149.044
C02958=1216.101,-72.827,-38.588,179.667,5.405,149.044
C02959=1216.096,-72.578,-38.599,179.670,5.406,149.043
C02960=1216.091,-72.328,-38.611,179.672,5.406,149.042
C02961=1216.086,-72.078,-38.622,179.674,5.406,149.042
C02962=1216.080,-71.829,-38.634,179.676,5.406,149.041
C02963=1216.075,-71.578,-38.645,179.679,5.406,149.040
C02964=1216.069,-71.329,-38.656,179.682,5.407,149.040
C02965=1216.065,-71.079,-38.668,179.684,5.406,149.039
C02966=1216.060,-70.830,-38.679,179.687,5.407,149.038
C02967=1216.055,-70.580,-38.691,179.689,5.406,149.037
C02968=1216.049,-70.331,-38.702,179.691,5.407,149.037
C02969=1216.044,-70.081,-38.714,179.693,5.407,149.036
C02970=1216.039,-69.831,-38.725,179.696,5.407,149.036
C02971=1216.034,-69.581,-38.737,179.698,5.408,149.035
C02972=1216.029,-69.332,-38.748,179.700,5.407,149.034
C02973=1216.024,-69.082,-38.760,179.703,5.408,149.033
C02974=1216.018,-68.833,-38.771,179.705,5.408,149.033
C02975=1216.013,-68.582,-38.782,179.708,5.408,149.032
C02976=1216.008,-68.333,-38.793,179.710,5.408,149.031
C02977=1216.002,-68.083,-38.805,179.713,5.408,149.031
C02978=1215.998,-67.833,-38.816,179.715,5.408,149.030
C02979=1215.992,-67.584,-38.828,179.717,5.408,149.029
C02980=1215.987,-67.334,-38.839,179.720,5.409,149.029
C02981=1215.982,-67.084,-38.851,179.722,5.409,149.028
C02982=1215.977,-66.835,-38.862,179.724,5.409,149.027
C02983=1215.972,-66.585,-38.874,179.726,5.409,149.027
C02984=1215.966,-66.335,-38.886,179.729,5.409,149.026
C02985=1215.961,-66.085,-38.898,179.732,5.410,149.025
C02986=1215.956,-65.837,-38.910,179.734,5.409,149.025
C02987=1215.951,-65.587,-38.921,179.736,5.410,149.024
C02988=1215.946,-65.337,-38.933,179.738,5.409,149.023
C02989=1215.941,-65.087,-38.944,179.741,5.410,149.022
C02990=1215.935,-64.838,-38.956,179.743,5.410,149.022
C02991=1215.930,-64.588,-38.968,179.746,5.410,149.021
C02992=1215.925,-64.338,-38.979,179.749,5.411,149.020
C02993=1215.920,-64.088,-38.991,179.751,5.410,149.020
C02994=1215.915,-63.839,-39.002,179.753,5.411,149.019
C02995=1215.909,-63.589,-39.014,179.755,5.411,149.018
C02996=1215.904,-63.339,-39.026,179.758,5.411,149.018
C02997=1215.899,-63.090,-39.037,179.760,5.411,149.017
C02998=1215.894,-62.840,-39.050,179.762,5.411,149.016
C02999=1215.889,-62.591,-39.061,179.765,5.412,149.016
C03000=1215.884,-62.341,-39.073,179.767,5.411,149.015
C03001=1215.878,-62.091,-39.085,179.770,5.412,149.014
C03002=1215.874,-61.841,-39.096,179.772,5.411,149.013
C03003=1215.868,-61.591,-39.108,179.775,5.412,149.013
C03004=1215.862,-61.342,-39.120,179.777,5.412,149.012
C03005=1215.858,-61.093,-39.132,179.779,5.412,149.011
C03006=1215.852,-60.843,-39.143,179.781,5.413,149.011
C03007=1215.847,-60.593,-39.155,179.784,5.412,149.010
C03008=1215.842,-60.343,-39.167,179.786,5.413,149.009
C03009=1215.837,-60.094,-39.178,179.789,5.413,149.009
C03010=1215.832,-59.844,-39.191,179.791,5.413,149.008
C03011=1215.827,-59.595,-39.202,179.794,5.414,149.007
C03012=1215.822,-59.345,-39.214,179.796,5.413,149.007
C03013=1215.816,-59.095,-39.226,179.798,5.414,149.006
C03014=1215.811,-58.845,-39.237,179.800,5.413,149.005
C03015=1215.806,-58.596,-39.250,179.803,5.414,149.005
C03016=1215.801,-58.346,-39.262,179.806,5.414,149.004
C03017=1215.796,-58.096,-39.273,179.808,5.414,149.003
C03018=1215.791,-57.847,-39.286,179.811,5.414,149.002
C03019=1215.786,-57.597,-39.298,179.813,5.414,149.002
C03020=1215.780,-57.347,-39.310,179.815,5.415,149.001
C03021=1215.776,-57.097,-39.321,179.818,5.415,149.001
C03022=1215.770,-56.848,-39.333,179.820,5.415,149.000
C03023=1215.765,-56.598,-39.345,179.822,5.415,148.999
C03024=1215.760,-56.348,-39.357,179.824,5.415,148.998
C03025=1215.755,-56.099,-39.369,179.827,5.416,148.998
C03026=1215.750,-55.849,-39.381,179.830,5.416,148.997
C03027=1215.744,-55.599,-39.393,179.832,5.416,148.996
C03028=1215.739,-55.350,-39.406,179.834,5.416,148.996
C03029=1215.735,-55.100,-39.417,179.837,5.417,148.995
C03030=1215.729,-54.850,-39.429,179.839,5.416,148.994
C03031=1215.724,-54.601,-39.441,179.842,5.417,148.993
C03032=1215.719,-54.351,-39.453,179.844,5.416,148.993
C03033=1215.714,-54.102,-39.465,179.847,5.417,148.992
C03034=1215.709,-53.852,-39.477,179.849,5.418,148.992
C03035=1215.703,-53.602,-39.489,179.851,5.417,148.991
C03036=1215.698,-53.353,-39.502,179.854,5.418,148.990
C03037=1215.693,-53.103,-39.514,179.856,5.417,148.989
C03038=1215.688,-52.853,-39.525,179.858,5.418,148.989
C03039=1215.683,-52.604,-39.537,179.861,5.418,148.988
C03040=1215.677,-52.354,-39.549,179.863,5.418,148.987
C03041=1215.672,-52.105,-39.562,179.866,5.418,148.987
C03042=1215.667,-51.855,-39.574,179.868,5.418,148.986
C03043=1215.662,-51.606,-39.586,179.870,5.419,148.985
C03044=1215.657,-51.356,-39.598,179.873,5.419,148.985
C03045=1215.652,-51.107,-39.610,179.875,5.419,148.984
C03046=1215.647,-50.857,-39.622,179.878,5.419,148.983
C03047=1215.642,-50.606,-39.634,179.881,5.420,148.982
C03048=1215.637,-50.357,-39.647,179.883,5.419,148.982
C03049=1215.631,-50.107,-39.659,179.885,5.420,148.981
C03050=1215.626,-49.858,-39.672,179.887,5.420,148.981
C03051=1215.621,-49.608,-39.683,179.890,5.420,148.980
C03052=1215.616,-49.359,-39.695,179.892,5.421,148.979
C03053=1215.610,-49.088,-39.709,179.894,5.420,148.978
C03054=1215.605,-48.819,-39.722,179.897,5.421,148.978
C03055=1215.599,-48.549,-39.735,179.900,5.421,148.977
C03056=1215.594,-48.278,-39.748,179.903,5.421,148.976
C03057=1215.589,-48.029,-39.761,179.905,5.421,148.975
C03058=1215.584,-47.780,-39.773,179.908,5.422,148.975
C03059=1215.578,-47.530,-39.785,179.910,5.422,148.974
C03060=1215.573,-47.280,-39.798,179.912,5.422,148.973
C03061=1215.568,-47.030,-39.810,179.915,5.422,148.973
C03062=1215.563,-46.781,-39.822,179.917,5.422,148.972
C03063=1215.557,-46.532,-39.835,179.920,5.422,148.971
C03064=1215.552,-46.282,-39.847,179.922,5.423,148.971
C03065=1215.548,-46.032,-39.860,179.924,5.423,148.970
C03066=1215.542,-45.782,-39.872,179.927,5.423,148.969
C03067=1215.537,-45.533,-39.884,179.929,5.424,148.969
C03068=1215.532,-45.283,-39.897,179.931,5.423,148.968
C03069=1215.526,-45.033,-39.909,179.934,5.424,148.967
C03070=1215.521,-44.784,-39.921,179.937,5.424,148.967
C03071=1215.516,-44.535,-39.934,179.939,5.424,148.966
C03072=1215.511,-44.284,-39.946,179.941,5.425,148.965
C03073=1215.506,-44.035,-39.959,179.944,5.424,148.964
C03074=1215.501,-43.785,-39.971,179.946,5.425,148.964
C03075=1215.496,-43.535,-39.983,179.949,5.425,148.963
C03076=1215.491,-43.286,-39.996,179.951,5.425,148.962
C03077=1215.485,-43.037,-40.009,179.954,5.425,148.962
C03078=1215.481,-42.786,-40.021,179.956,5.426,148.961
C03079=1215.475,-42.537,-40.033,179.958,5.425,148.960
C03080=1215.470,-42.288,-40.046,179.961,5.426,148.960
C03081=1215.465,-42.038,-40.058,179.963,5.427,148.959
C03082=1215.460,-41.788,-40.070,179.965,5.426,148.958
C03083=1215.455,-41.538,-40.083,179.968,5.427,148.958
C03084=1215.450,-41.289,-40.096,179.971,5.427,148.957
C03085=1215.445,-41.039,-40.108,179.973,5.427,148.956
C03086=1215.440,-40.790,-40.121,179.975,5.427,148.956
C03087=1215.434,-40.540,-40.133,179.978,5.428,148.955
C03088=1215.429,-40.290,-40.147,179.980,5.428,148.954
C03089=1215.424,-40.041,-40.159,179.983,5.428,148.953
C03090=1215.419,-39.791,-40.171,179.985,5.428,148.953
C03091=1215.414,-39.541,-40.184,179.987,5.428,148.952
C03092=1215.408,-39.292,-40.196,179.990,5.429,148.951
C03093=1215.404,-39.042,-40.209,179.992,5.428,148.951
C03094=1215.399,-38.793,-40.222,179.995,5.429,148.950
C03095=1215.393,-38.543,-40.234,179.998,5.429,148.949
C03096=1215.388,-38.294,-40.246,180.000,5.429,148.949
C03097=1215.383,-38.043,-40.260,-179.998,5.430,148.948
C03098=1215.378,-37.794,-40.273,-179.996,5.430,148.947
C03099=1215.373,-37.545,-40.285,-179.993,5.430,148.947
C03100=1215.368,-37.295,-40.298,-179.991,5.431,148.946
C03101=1215.363,-37.045,-40.311,-179.988,5.431,148.945
C03102=1215.358,-36.795,-40.323,-179.986,5.431,148.945
C03103=1215.352,-36.546,-40.336,-179.983,5.431,148.944
C03104=1215.347,-36.296,-40.348,-179.981,5.432,148.943
C03105=1215.342,-36.046,-40.361,-179.979,5.431,148.942
C03106=1215.337,-35.797,-40.374,-179.976,5.432,148.942
C03107=1215.332,-35.548,-40.387,-179.973,5.432,148.941
C03108=1215.327,-35.298,-40.399,-179.971,5.432,148.940
C03109=1215.321,-35.048,-40.413,-179.969,5.432,148.940
C03110=1215.316,-34.799,-40.425,-179.966,5.433,148.939
C03111=1215.311,-34.549,-40.438,-179.964,5.433,148.938
C03112=1215.307,-34.299,-40.451,-179.961,5.433,148.938
C03113=1215.301,-34.050,-40.464,-179.958,5.433,148.937
C03114=1215.296,-33.800,-40.477,-179.957,5.434,148.936
C03115=1215.291,-33.550,-40.490,-179.954,5.434,148.936
C03116=1215.286,-33.301,-40.502,-179.952,5.435,148.935
C03117=1215.281,-33.052,-40.515,-179.949,5.434,148.934
C03118=1215.275,-32.802,-40.528,-179.947,5.435,148.934
C03119=1215.271,-32.552,-40.541,-179.944,5.435,148.933
C03120=1215.265,-32.303,-40.554,-179.942,5.435,148.932
C03121=1215.260,-32.053,-40.567,-179.939,5.435,148.932
C03122=1215.255,-31.803,-40.580,-179.937,5.436,148.931
C03123=1215.250,-31.554,-40.592,-179.934,5.436,148.930
C03124=1215.245,-31.305,-40.605,-179.932,5.436,148.929
C03125=1215.240,-31.054,-40.619,-179.929,5.436,148.929
C03126=1215.234,-30.805,-40.631,-179.927,5.437,148.928
C03127=1215.229,-30.556,-40.644,-179.925,5.437,148.927
C03128=1215.225,-30.306,-40.657,-179.922,5.437,148.927
C03129=1215.219,-30.056,-40.670,-179.919,5.438,148.926
C03130=1215.214,-29.806,-40.683,-179.917,5.437,148.925
C03131=1215.209,-29.557,-40.696,-179.915,5.438,148.925
C03132=1215.203,-29.307,-40.709,-179.912,5.439,148.924
C03133=1215.199,-29.057,-40.722,-179.910,5.438,148.923
C03134=1215.194,-28.808,-40.735,-179.908,5.439,148.923
C03135=1215.188,-28.559,-40.748,-179.905,5.439,148.922
C03136=1215.184,-28.309,-40.761,-179.903,5.439,148.921
C03137=1215.179,-28.059,-40.774,-179.900,5.439,148.921
C03138=1215.173,-27.809,-40.787,-179.898,5.440,148.920
C03139=1215.168,-27.560,-40.800,-179.895,5.440,148.919
C03140=1215.163,-27.310,-40.813,-179.893,5.440,148.918
C03141=1215.158,-27.061,-40.827,-179.890,5.441,148.918
C03142=1215.153,-26.811,-40.839,-179.888,5.441,148.917
C03143=1215.148,-26.561,-40.853,-179.885,5.441,148.916
C03144=1215.143,-26.312,-40.866,-179.883,5.441,148.916
C03145=1215.137,-26.062,-40.878,-179.880,5.442,148.915
C03146=1215.133,-25.813,-40.892,-179.878,5.441,148.914
C03147=1215.127,-25.563,-40.905,-179.875,5.442,148.914
C03148=1215.122,-25.313,-40.919,-179.873,5.442,148.913
C03149=1215.117,-25.064,-40.931,-179.871,5.443,148.912
C03150=1215.113,-24.814,-40.945,-179.868,5.443,148.912
C03151=1215.107,-24.565,-40.958,-179.866,5.443,148.911
C03152=1215.102,-24.315,-40.971,-179.863,5.444,148.910
C03153=1215.097,-24.065,-40.984,-179.861,5.443,148.910
C03154=1215.092,-23.816,-40.998,-179.858,5.444,148.909
C03155=1215.087,-23.566,-41.011,-179.856,5.444,148.908
C03156=1215.081,-23.317,-41.024,-179.854,5.444,148.908
C03157=1215.076,-23.047,-41.039,-179.851,5.445,148.907
C03158=1215.071,-22.777,-41.052,-179.848,5.445,148.906
C03159=1215.065,-22.509,-41.067,-179.845,5.445,148.905
C03160=1215.059,-22.239,-41.081,-179.843,5.446,148.905
C03161=1215.055,-21.989,-41.094,-179.840,5.446,148.904
C03162=1215.050,-21.740,-41.108,-179.838,5.446,148.903
C03163=1215.045,-21.490,-41.121,-179.835,5.446,148.902
C03164=1215.039,-21.240,-41.134,-179.833,5.447,148.902
C03165=1215.034,-20.991,-41.148,-179.831,5.447,148.901
C03166=1215.029,-20.741,-41.161,-179.828,5.447,148.901
C03167=1215.024,-20.492,-41.175,-179.826,5.448,148.900
C03168=1215.019,-20.242,-41.188,-179.823,5.448,148.899
C03169=1215.013,-19.993,-41.201,-179.821,5.448,148.899
C03170=1215.008,-19.743,-41.215,-179.818,5.449,148.898
C03171=1215.003,-19.494,-41.228,-179.816,5.449,148.897
C03172=1214.998,-19.244,-41.242,-179.813,5.449,148.896
C03173=1214.993,-18.995,-41.254,-179.811,5.449,148.896
C03174=1214.988,-18.744,-41.268,-179.808,5.450,148.895
C03175=1214.984,-18.495,-41.282,-179.805,5.450,148.894
C03176=1214.978,-18.245,-41.295,-179.803,5.450,148.894
C03177=1214.974,-17.996,-41.309,-179.801,5.450,148.893
C03178=1214.968,-17.746,-41.322,-179.798,5.451,148.892
C03179=1214.963,-17.497,-41.336,-179.795,5.451,148.892
C03180=1214.958,-17.247,-41.349,-179.794,5.451,148.891
C03181=1214.953,-16.998,-41.363,-179.791,5.452,148.890
C03182=1214.948,-16.748,-41.376,-179.789,5.452,148.890
C03183=1214.943,-16.498,-41.390,-179.786,5.453,148.889
C03184=1214.937,-16.249,-41.403,-179.784,5.453,148.888
C03185=1214.933,-15.999,-41.417,-179.781,5.453,148.888
C03186=1214.927,-15.750,-41.430,-179.778,5.454,148.887
C03187=1214.923,-15.500,-41.444,-179.776,5.453,148.886
C03188=1214.917,-15.250,-41.457,-179.774,5.454,148.886
C03189=1214.912,-15.001,-41.471,-179.771,5.454,148.885
C03190=1214.907,-14.751,-41.484,-179.768,5.455,148.884
C03191=1214.902,-14.502,-41.498,-179.766,5.454,148.883
C03192=1214.896,-14.252,-41.511,-179.764,5.455,148.883
C03193=1214.892,-14.003,-41.525,-179.761,5.455,148.882
C03194=1214.887,-13.753,-41.539,-179.758,5.456,148.881
C03195=1214.881,-13.503,-41.553,-179.757,5.456,148.881
C03196=1214.877,-13.254,-41.566,-179.754,5.457,148.880
C03197=1214.871,-13.004,-41.580,-179.751,5.457,148.880
C03198=1214.866,-12.755,-41.593,-179.749,5.458,148.879
C03199=1214.862,-12.506,-41.607,-179.747,5.457,148.878
C03200=1214.856,-12.255,-41.621,-179.744,5.458,148.877
C03201=1214.851,-12.006,-41.635,-179.741,5.458,148.877
C03202=1214.846,-11.756,-41.648,-179.739,5.459,148.876
C03203=1214.841,-11.506,-41.662,-179.737,5.458,148.875
C03204=1214.836,-11.257,-41.676,-179.734,5.459,148.875
C03205=1214.831,-11.007,-41.689,-179.731,5.459,148.874
C03206=1214.826,-10.758,-41.703,-179.729,5.460,148.873
C03207=1214.821,-10.509,-41.717,-179.727,5.460,148.873
C03208=1214.815,-10.258,-41.730,-179.724,5.460,148.872
C03209=1214.811,-10.010,-41.744,-179.721,5.461,148.871
C03210=1214.806,-9.760,-41.758,-179.719,5.461,148.871
C03211=1214.801,-9.510,-41.772,-179.717,5.461,148.870
C03212=1214.795,-9.261,-41.786,-179.714,5.462,148.869
C03213=1214.791,-9.011,-41.799,-179.712,5.462,148.869
C03214=1214.786,-8.762,-41.813,-179.709,5.463,148.868
C03215=1214.780,-8.512,-41.827,-179.706,5.463,148.867
C03216=1214.775,-8.262,-41.841,-179.704,5.463,148.867
C03217=1214.771,-8.013,-41.855,-179.702,5.463,148.866
C03218=1214.765,-7.764,-41.869,-179.699,5.464,148.865
C03219=1214.760,-7.514,-41.883,-179.696,5.464,148.865
C03220=1214.755,-7.264,-41.896,-179.694,5.464,148.864
C03221=1214.749,-7.015,-41.910,-179.692,5.465,148.863
C03222=1214.745,-6.765,-41.924,-179.689,5.465,148.862
C03223=1214.740,-6.516,-41.938,-179.686,5.466,148.862
C03224=1214.735,-6.266,-41.953,-179.685,5.466,148.861
C03225=1214.729,-6.016,-41.966,-179.682,5.466,148.861
C03226=1214.724,-5.767,-41.980,-179.679,5.467,148.860
C03227=1214.719,-5.517,-41.994,-179.677,5.467,148.859
C03228=1214.715,-5.268,-42.008,-179.674,5.468,148.859
C03229=1214.710,-5.018,-42.022,-179.672,5.467,148.858
C03230=1214.705,-4.769,-42.036,-179.669,5.468,148.857
C03231=1214.699,-4.518,-42.050,-179.667,5.468,148.856
C03232=1214.694,-4.269,-42.064,-179.664,5.469,148.856
C03233=1214.689,-4.020,-42.078,-179.662,5.469,148.855
C03234=1214.684,-3.770,-42.092,-179.659,5.469,148.854
C03235=1214.679,-3.521,-42.105,-179.657,5.470,148.854
C03236=1214.674,-3.272,-42.120,-179.654,5.470,148.853
C03237=1214.669,-3.022,-42.134,-179.652,5.471,148.853
C03238=1214.664,-2.772,-42.148,-179.650,5.471,148.852
C03239=1214.659,-2.523,-42.162,-179.647,5.471,148.851
C03240=1214.654,-2.273,-42.177,-179.645,5.472,148.851
C03241=1214.649,-2.024,-42.191,-179.642,5.472,148.850
C03242=1214.643,-1.773,-42.204,-179.639,5.473,148.849
C03243=1214.638,-1.524,-42.218,-179.637,5.472,148.848
C03244=1214.633,-1.275,-42.233,-179.635,5.473,148.848
C03245=1214.628,-1.025,-42.247,-179.632,5.473,148.847
C03246=1214.623,-0.775,-42.261,-179.629,5.474,148.846
C03247=1214.618,-0.526,-42.275,-179.627,5.474,148.846
C03248=1214.613,-0.277,-42.289,-179.624,5.474,148.845
C03249=1214.608,-0.027,-42.303,-179.622,5.475,148.844
C03250=1214.603,0.223,-42.317,-179.620,5.475,148.844
C03251=1214.598,0.472,-42.332,-179.617,5.476,148.843
C03252=1214.593,0.722,-42.346,-179.614,5.476,148.842
C03253=1214.588,0.971,-42.360,-179.612,5.476,148.842
C03254=1214.583,1.221,-42.374,-179.610,5.477,148.841
C03255=1214.578,1.470,-42.389,-179.607,5.477,148.840
C03256=1214.573,1.719,-42.403,-179.604,5.478,148.840
C03257=1214.568,1.969,-42.418,-179.602,5.478,148.839
C03258=1214.563,2.218,-42.431,-179.600,5.478,148.838
C03259=1214.558,2.468,-42.446,-179.597,5.478,148.838
C03260=1214.553,2.718,-42.460,-179.594,5.479,148.837
C03261=1214.547,2.987,-42.476,-179.592,5.479,148.836
C03262=1214.542,3.256,-42.491,-179.589,5.480,148.836
C03263=1214.537,3.525,-42.507,-179.586,5.480,148.835
C03264=1214.531,3.794,-42.522,-179.584,5.481,148.834
C03265=1214.526,4.043,-42.536,-179.581,5.482,148.834
C03266=1214.521,4.292,-42.551,-179.579,5.481,148.833
C03267=1214.516,4.542,-42.565,-179.576,5.482,148.832
C03268=1214.511,4.792,-42.579,-179.574,5.482,148.831
C03269=1214.506,5.042,-42.594,-179.571,5.483,148.831
C03270=1214.501,5.291,-42.608,-179.568,5.483,148.830
C03271=1214.496,5.541,-42.622,-179.566,5.484,148.829
C03272=1214.491,5.789,-42.637,-179.564,5.484,148.829
C03273=1214.485,6.039,-42.652,-179.561,5.484,148.828
C03274=1214.480,6.289,-42.666,-179.559,5.485,148.828
C03275=1214.475,6.539,-42.680,-179.556,5.485,148.827
C03276=1214.470,6.789,-42.695,-179.553,5.486,148.826
C03277=1214.466,7.038,-42.710,-179.551,5.486,148.826
C03278=1214.461,7.287,-42.724,-179.549,5.486,148.825
C03279=1214.456,7.537,-42.738,-179.546,5.487,148.824
C03280=1214.451,7.787,-42.752,-179.543,5.487,148.823
C03281=1214.445,8.036,-42.768,-179.541,5.488,148.823
C03282=1214.440,8.285,-42.782,-179.538,5.488,148.822
C03283=1214.435,8.535,-42.796,-179.537,5.488,148.822
C03284=1214.430,8.785,-42.810,-179.534,5.489,148.821
C03285=1214.425,9.034,-42.825,-179.531,5.489,148.820
C03286=1214.420,9.283,-42.840,-179.529,5.490,148.820
C03287=1214.415,9.533,-42.854,-179.526,5.490,148.819
C03288=1214.410,9.783,-42.870,-179.523,5.491,148.818
C03289=1214.405,10.032,-42.884,-179.521,5.491,148.818
C03290=1214.400,10.282,-42.898,-179.519,5.491,148.817
C03291=1214.395,10.531,-42.913,-179.516,5.492,148.816
C03292=1214.390,10.781,-42.927,-179.513,5.492,148.815
C03293=1214.385,11.031,-42.942,-179.511,5.493,148.815
C03294=1214.380,11.280,-42.957,-179.508,5.493,148.814
C03295=1214.375,11.530,-42.972,-179.506,5.494,148.814
C03296=1214.371,11.779,-42.987,-179.504,5.494,148.813
C03297=1214.365,12.029,-43.001,-179.501,5.494,148.812
C03298=1214.360,12.278,-43.016,-179.498,5.495,148.812
C03299=1214.355,12.527,-43.030,-179.496,5.495,148.811
C03300=1214.350,12.776,-43.045,-179.493,5.496,148.810
C03301=1214.344,13.026,-43.060,-179.491,5.496,148.810
C03302=1214.339,13.276,-43.075,-179.488,5.496,148.809
C03303=1214.334,13.525,-43.089,-179.486,5.497,148.808
C03304=1214.330,13.774,-43.104,-179.484,5.497,148.808
C03305=1214.324,14.024,-43.119,-179.481,5.498,148.807
C03306=1214.319,14.274,-43.134,-179.478,5.498,148.806
C03307=1214.314,14.523,-43.148,-179.476,5.499,148.806
C03308=1214.310,14.772,-43.163,-179.473,5.500,148.805
C03309=1214.304,15.022,-43.178,-179.471,5.499,148.804
C03310=1214.299,15.271,-43.193,-179.468,5.500,148.804
C03311=1214.295,15.521,-43.207,-179.466,5.500,148.803
C03312=1214.289,15.771,-43.223,-179.464,5.501,148.802
C03313=1214.285,16.021,-43.237,-179.461,5.502,148.802
C03314=1214.280,16.270,-43.252,-179.458,5.502,148.801
C03315=1214.274,16.520,-43.267,-179.456,5.503,148.800
C03316=1214.270,16.769,-43.282,-179.453,5.503,148.800
C03317=1214.265,17.019,-43.296,-179.451,5.503,148.799
C03318=1214.259,17.268,-43.312,-179.448,5.503,148.798
C03319=1214.255,17.517,-43.327,-179.446,5.504,148.798
C03320=1214.250,17.767,-43.341,-179.443,5.505,148.797
C03321=1214.244,18.016,-43.357,-179.441,5.505,148.797
C03322=1214.239,18.266,-43.371,-179.438,5.506,148.796
C03323=1214.234,18.516,-43.387,-179.435,5.506,148.795
C03324=1214.229,18.765,-43.402,-179.433,5.507,148.795
C03325=1214.224,19.014,-43.416,-179.431,5.507,148.794
C03326=1214.219,19.264,-43.432,-179.428,5.507,148.793
C03327=1214.214,19.514,-43.446,-179.425,5.508,148.792
C03328=1214.209,19.763,-43.461,-179.423,5.508,148.792
C03329=1214.204,20.012,-43.476,-179.420,5.509,148.791
C03330=1214.200,20.262,-43.491,-179.418,5.510,148.791
C03331=1214.194,20.512,-43.507,-179.415,5.510,148.790
C03332=1214.190,20.761,-43.522,-179.413,5.511,148.789
C03333=1214.184,21.011,-43.537,-179.411,5.510,148.789
C03334=1214.179,21.260,-43.552,-179.408,5.511,148.788
C03335=1214.174,21.509,-43.567,-179.405,5.512,148.787
C03336=1214.169,21.759,-43.581,-179.403,5.512,148.787
C03337=1214.164,22.008,-43.596,-179.400,5.513,148.786
C03338=1214.159,22.258,-43.612,-179.398,5.513,148.785
C03339=1214.155,22.507,-43.627,-179.395,5.514,148.785
C03340=1214.149,22.757,-43.642,-179.393,5.515,148.784
C03341=1214.145,23.007,-43.657,-179.390,5.515,148.783
C03342=1214.139,23.256,-43.673,-179.387,5.516,148.783
C03343=1214.135,23.505,-43.688,-179.385,5.515,148.782
C03344=1214.129,23.755,-43.703,-179.383,5.516,148.781
C03345=1214.124,24.004,-43.718,-179.380,5.516,148.781
C03346=1214.119,24.254,-43.734,-179.378,5.517,148.780
C03347=1214.115,24.503,-43.749,-179.375,5.518,148.780
C03348=1214.109,24.753,-43.764,-179.372,5.518,148.779
C03349=1214.104,25.002,-43.778,-179.370,5.519,148.778
C03350=1214.099,25.252,-43.794,-179.367,5.519,148.777
C03351=1214.094,25.501,-43.809,-179.365,5.520,148.777
C03352=1214.089,25.750,-43.825,-179.362,5.520,148.776
C03353=1214.084,26.000,-43.841,-179.360,5.520,148.775
C03354=1214.080,26.250,-43.856,-179.358,5.521,148.775
C03355=1214.074,26.500,-43.870,-179.355,5.522,148.774
C03356=1214.069,26.749,-43.885,-179.352,5.522,148.774
C03357=1214.064,26.998,-43.901,-179.350,5.523,148.773
C03358=1214.060,27.248,-43.916,-179.347,5.523,148.772
C03359=1214.054,27.497,-43.932,-179.344,5.524,148.772
C03360=1214.049,27.747,-43.948,-179.342,5.524,148.771
C03361=1214.044,27.996,-43.963,-179.340,5.525,148.770
C03362=1214.039,28.245,-43.978,-179.337,5.526,148.770
C03363=1214.035,28.495,-43.994,-179.334,5.526,148.769
C03364=1214.030,28.744,-44.009,-179.332,5.527,148.768
C03365=1214.024,29.013,-44.025,-179.329,5.527,148.768
C03366=1214.019,29.282,-44.042,-179.326,5.528,148.767
C03367=1214.013,29.551,-44.058,-179.324,5.528,148.766
C03368=1214.007,29.819,-44.075,-179.321,5.529,148.766
C03369=1214.003,30.068,-44.090,-179.319,5.529,148.765
C03370=1213.998,30.318,-44.106,-179.316,5.530,148.764
C03371=1213.993,30.568,-44.122,-179.313,5.530,148.764
C03372=1213.988,30.817,-44.137,-179.311,5.531,148.763
C03373=1213.983,31.066,-44.152,-179.309,5.531,148.762
C03374=1213.978,31.316,-44.168,-179.306,5.532,148.762
C03375=1213.973,31.565,-44.183,-179.304,5.532,148.761
C03376=1213.968,31.815,-44.199,-179.301,5.533,148.761
C03377=1213.963,32.065,-44.215,-179.298,5.533,148.760
C03378=1213.958,32.314,-44.230,-179.296,5.534,148.759
C03379=1213.953,32.563,-44.245,-179.293,5.534,148.758
C03380=1213.948,32.813,-44.261,-179.290,5.535,148.758
C03381=1213.943,33.063,-44.277,-179.288,5.536,148.757
C03382=1213.938,33.311,-44.293,-179.286,5.536,148.757
C03383=1213.933,33.561,-44.308,-179.283,5.537,148.756
C03384=1213.928,33.811,-44.324,-179.280,5.537,148.755
C03385=1213.924,34.060,-44.339,-179.278,5.538,148.755
C03386=1213.918,34.309,-44.355,-179.275,5.538,148.754
C03387=1213.913,34.559,-44.370,-179.273,5.539,148.754
C03388=1213.908,34.809,-44.386,-179.270,5.540,148.753
C03389=1213.903,35.058,-44.401,-179.268,5.540,148.752
C03390=1213.898,35.307,-44.418,-179.265,5.541,148.752
C03391=1213.894,35.557,-44.433,-179.263,5.541,148.751
C03392=1213.888,35.806,-44.449,-179.260,5.541,148.750
C03393=1213.883,36.056,-44.465,-179.258,5.542,148.749
C03394=1213.879,36.306,-44.480,-179.256,5.543,148.749
C03395=1213.873,36.555,-44.496,-179.253,5.543,148.748
C03396=1213.868,36.804,-44.512,-179.250,5.544,148.748
C03397=1213.863,37.054,-44.528,-179.248,5.544,148.747
C03398=1213.858,37.303,-44.543,-179.245,5.545,148.746
C03399=1213.853,37.552,-44.558,-179.242,5.545,148.746
C03400=1213.849,37.802,-44.574,-179.240,5.546,148.745
C03401=1213.844,38.051,-44.591,-179.238,5.547,148.745
C03402=1213.838,38.301,-44.606,-179.235,5.547,148.744
C03403=1213.833,38.551,-44.622,-179.232,5.548,148.743
C03404=1213.828,38.799,-44.639,-179.230,5.548,148.743
C03405=1213.824,39.050,-44.654,-179.227,5.549,148.742
C03406=1213.819,39.299,-44.669,-179.225,5.550,148.741
C03407=1213.814,39.548,-44.685,-179.222,5.550,148.741
C03408=1213.809,39.798,-44.702,-179.220,5.551,148.740
C03409=1213.804,40.047,-44.717,-179.217,5.551,148.739
C03410=1213.798,40.296,-44.733,-179.214,5.552,148.739
C03411=1213.794,40.546,-44.750,-179.212,5.553,148.738
C03412=1213.788,40.795,-44.765,-179.209,5.553,148.738
C03413=1213.784,41.045,-44.781,-179.207,5.554,148.737
C03414=1213.779,41.294,-44.797,-179.204,5.555,148.736
C03415=1213.774,41.544,-44.813,-179.202,5.555,148.736
C03416=1213.769,41.793,-44.828,-179.199,5.556,148.735
C03417=1213.764,42.042,-44.845,-179.196,5.556,148.734
C03418=1213.759,42.292,-44.861,-179.194,5.557,148.734
C03419=1213.754,42.541,-44.877,-179.191,5.558,148.733
C03420=1213.749,42.791,-44.893,-179.189,5.558,148.732
C03421=1213.744,43.041,-44.908,-179.186,5.559,148.732
C03422=1213.739,43.289,-44.925,-179.184,5.559,148.731
C03423=1213.734,43.539,-44.941,-179.181,5.560,148.731
C03424=1213.729,43.788,-44.957,-179.179,5.561,148.730
C03425=1213.724,44.038,-44.973,-179.176,5.561,148.729
C03426=1213.719,44.287,-44.989,-179.174,5.562,148.729
C03427=1213.714,44.537,-45.005,-179.171,5.562,148.728
C03428=1213.709,44.787,-45.021,-179.168,5.563,148.727
C03429=1213.705,45.036,-45.038,-179.166,5.564,148.727
C03430=1213.699,45.285,-45.053,-179.163,5.564,148.726
C03431=1213.695,45.535,-45.070,-179.161,5.565,148.726
C03432=1213.689,45.784,-45.085,-179.158,5.565,148.725
C03433=1213.685,46.034,-45.102,-179.156,5.566,148.724
C03434=1213.679,46.283,-45.118,-179.153,5.567,148.724
C03435=1213.675,46.533,-45.134,-179.151,5.567,148.723
C03436=1213.670,46.782,-45.151,-179.148,5.568,148.722
C03437=1213.665,47.032,-45.167,-179.145,5.569,148.722
C03438=1213.660,47.280,-45.183,-179.143,5.569,148.721
C03439=1213.655,47.531,-45.199,-179.141,5.570,148.721
C03440=1213.650,47.779,-45.215,-179.138,5.571,148.720
C03441=1213.645,48.029,-45.231,-179.135,5.571,148.719
C03442=1213.640,48.278,-45.247,-179.133,5.572,148.719
C03443=1213.636,48.528,-45.264,-179.130,5.572,148.718
C03444=1213.630,48.777,-45.280,-179.128,5.573,148.717
C03445=1213.625,49.027,-45.297,-179.125,5.574,148.717
C03446=1213.620,49.276,-45.312,-179.123,5.574,148.716
C03447=1213.615,49.526,-45.329,-179.120,5.575,148.715
C03448=1213.610,49.775,-45.345,-179.117,5.575,148.715
C03449=1213.605,50.025,-45.361,-179.115,5.576,148.714
C03450=1213.600,50.273,-45.378,-179.113,5.577,148.714
C03451=1213.596,50.523,-45.394,-179.110,5.577,148.713
C03452=1213.591,50.773,-45.410,-179.107,5.578,148.712
C03453=1213.586,51.022,-45.427,-179.105,5.578,148.712
C03454=1213.581,51.272,-45.444,-179.103,5.579,148.711
C03455=1213.575,51.521,-45.459,-179.100,5.580,148.711
C03456=1213.571,51.770,-45.476,-179.097,5.580,148.710
C03457=1213.566,52.019,-45.492,-179.095,5.581,148.709
C03458=1213.561,52.269,-45.509,-179.092,5.582,148.709
C03459=1213.557,52.519,-45.525,-179.090,5.582,148.708
C03460=1213.551,52.768,-45.542,-179.087,5.583,148.707
C03461=1213.546,53.017,-45.559,-179.085,5.584,148.707
C03462=1213.541,53.266,-45.575,-179.082,5.584,148.706
C03463=1213.536,53.516,-45.591,-179.079,5.585,148.705
C03464=1213.532,53.766,-45.608,-179.077,5.586,148.705
C03465=1213.526,54.015,-45.624,-179.075,5.586,148.704
C03466=1213.522,54.264,-45.641,-179.072,5.587,148.704
C03467=1213.516,54.514,-45.657,-179.069,5.587,148.703
C03468=1213.512,54.763,-45.673,-179.067,5.589,148.703
C03469=1213.506,55.031,-45.692,-179.064,5.590,148.702
C03470=1213.501,55.300,-45.710,-179.061,5.590,148.701
C03471=1213.496,55.568,-45.727,-179.059,5.591,148.701
C03472=1213.491,55.837,-45.745,-179.056,5.591,148.700
C03473=1213.485,56.086,-45.762,-179.053,5.592,148.699
C03474=1213.481,56.336,-45.779,-179.051,5.592,148.699
C03475=1213.476,56.585,-45.795,-179.048,5.594,148.698
C03476=1213.470,56.835,-45.811,-179.045,5.595,148.697
C03477=1213.465,57.084,-45.828,-179.043,5.595,148.697
C03478=1213.461,57.334,-45.845,-179.040,5.596,148.696
C03479=1213.456,57.583,-45.861,-179.038,5.596,148.695
C03480=1213.451,57.832,-45.878,-179.035,5.597,148.695
C03481=1213.446,58.082,-45.895,-179.033,5.598,148.694
C03482=1213.441,58.331,-45.911,-179.030,5.598,148.694
C03483=1213.436,58.580,-45.928,-179.027,5.599,148.693
C03484=1213.431,58.830,-45.945,-179.025,5.599,148.692
C03485=1213.426,59.079,-45.961,-179.023,5.600,148.692
C03486=1213.421,59.328,-45.979,-179.020,5.601,148.691
C03487=1213.417,59.578,-45.995,-179.017,5.601,148.691
C03488=1213.412,59.827,-46.012,-179.015,5.602,148.690
C03489=1213.406,60.077,-46.029,-179.013,5.603,148.690
C03490=1213.402,60.326,-46.046,-179.009,5.604,148.689
C03491=1213.397,60.575,-46.062,-179.007,5.605,148.688
C03492=1213.392,60.825,-46.079,-179.004,5.605,148.688
C03493=1213.387,61.074,-46.096,-179.002,5.606,148.687
C03494=1213.382,61.324,-46.113,-178.999,5.607,148.686
C03495=1213.377,61.573,-46.129,-178.997,5.607,148.686
C03496=1213.372,61.822,-46.146,-178.994,5.608,148.685
C03497=1213.367,62.072,-46.163,-178.992,5.609,148.684
C03498=1213.363,62.321,-46.180,-178.989,5.610,148.684
C03499=1213.357,62.571,-46.197,-178.987,5.610,148.683
C03500=1213.352,62.820,-46.214,-178.984,5.611,148.683
C03501=1213.348,63.069,-46.230,-178.981,5.611,148.682
C03502=1213.343,63.319,-46.248,-178.979,5.613,148.682
C03503=1213.338,63.567,-46.265,-178.976,5.613,148.681
C03504=1213.333,63.817,-46.282,-178.973,5.614,148.680
C03505=1213.328,64.067,-46.298,-178.971,5.615,148.680
C03506=1213.323,64.317,-46.316,-178.969,5.616,148.679
C03507=1213.318,64.565,-46.332,-178.966,5.616,148.678
C03508=1213.313,64.815,-46.349,-178.963,5.617,148.678
C03509=1213.308,65.065,-46.366,-178.961,5.617,148.677
C03510=1213.303,65.314,-46.384,-178.959,5.618,148.677
C03511=1213.299,65.563,-46.401,-178.956,5.619,148.676
C03512=1213.293,65.812,-46.418,-178.953,5.620,148.675
C03513=1213.288,66.062,-46.434,-178.951,5.621,148.675
C03514=1213.283,66.312,-46.451,-178.948,5.622,148.674
C03515=1213.279,66.560,-46.469,-178.945,5.622,148.674
C03516=1213.274,66.810,-46.486,-178.943,5.623,148.673
C03517=1213.269,67.059,-46.502,-178.941,5.624,148.673
C03518=1213.264,67.309,-46.520,-178.938,5.624,148.672
C03519=1213.259,67.558,-46.537,-178.935,5.625,148.671
C03520=1213.254,67.808,-46.554,-178.933,5.625,148.671
C03521=1213.250,68.057,-46.571,-178.930,5.627,148.670
C03522=1213.244,68.306,-46.588,-178.927,5.628,148.669
C03523=1213.240,68.555,-46.605,-178.925,5.628,148.669
C03524=1213.234,68.805,-46.623,-178.922,5.629,148.668
C03525=1213.229,69.055,-46.640,-178.920,5.630,148.668
C03526=1213.225,69.303,-46.657,-178.917,5.630,148.667
C03527=1213.220,69.553,-46.674,-178.915,5.631,148.666
C03528=1213.215,69.803,-46.691,-178.913,5.632,148.666
C03529=1213.210,70.051,-46.709,-178.910,5.632,148.665
C03530=1213.205,70.301,-46.725,-178.907,5.634,148.665
C03531=1213.200,70.550,-46.743,-178.904,5.634,148.664
C03532=1213.195,70.800,-46.761,-178.902,5.635,148.664
C03533=1213.191,71.049,-46.777,-178.899,5.636,148.663
C03534=1213.186,71.298,-46.795,-178.897,5.636,148.662
C03535=1213.181,71.548,-46.813,-178.895,5.637,148.662
C03536=1213.176,71.798,-46.829,-178.892,5.638,148.661
C03537=1213.171,72.046,-46.847,-178.889,5.639,148.660
C03538=1213.165,72.296,-46.864,-178.886,5.640,148.660
C03539=1213.161,72.545,-46.882,-178.884,5.641,148.659
C03540=1213.156,72.794,-46.899,-178.881,5.641,148.659
C03541=1213.151,73.044,-46.916,-178.879,5.642,148.658
C03542=1213.147,73.293,-46.933,-178.877,5.643,148.658
C03543=1213.141,73.543,-46.951,-178.874,5.643,148.657
C03544=1213.137,73.792,-46.969,-178.871,5.645,148.656
C03545=1213.132,74.042,-46.985,-178.868,5.645,148.656
C03546=1213.127,74.291,-47.003,-178.866,5.646,148.655
C03547=1213.122,74.541,-47.021,-178.863,5.647,148.655
C03548=1213.117,74.789,-47.038,-178.861,5.647,148.654
C03549=1213.112,75.039,-47.055,-178.859,5.648,148.654
C03550=1213.107,75.288,-47.073,-178.856,5.649,148.653
C03551=1213.102,75.537,-47.090,-178.853,5.650,148.652
C03552=1213.098,75.786,-47.108,-178.850,5.651,148.652
C03553=1213.093,76.036,-47.125,-178.848,5.652,148.651
C03554=1213.088,76.285,-47.143,-178.845,5.652,148.650
C03555=1213.083,76.535,-47.161,-178.843,5.653,148.650
C03556=1213.078,76.784,-47.177,-178.841,5.654,148.649
C03557=1213.073,77.033,-47.195,-178.837,5.655,148.649
C03558=1213.068,77.282,-47.213,-178.835,5.656,148.648
C03559=1213.063,77.532,-47.231,-178.833,5.657,148.648
C03560=1213.059,77.781,-47.248,-178.830,5.657,148.647
C03561=1213.054,78.031,-47.265,-178.827,5.658,148.646
C03562=1213.049,78.280,-47.283,-178.825,5.659,148.646
C03563=1213.044,78.529,-47.301,-178.822,5.660,148.645
C03564=1213.039,78.779,-47.318,-178.820,5.661,148.645
C03565=1213.034,79.028,-47.336,-178.817,5.661,148.644
C03566=1213.030,79.277,-47.354,-178.815,5.662,148.643
C03567=1213.024,79.527,-47.371,-178.812,5.663,148.643
C03568=1213.019,79.776,-47.389,-178.809,5.663,148.642
C03569=1213.015,80.025,-47.407,-178.807,5.665,148.642
C03570=1213.009,80.275,-47.424,-178.804,5.666,148.641
C03571=1213.004,80.524,-47.442,-178.802,5.666,148.640
C03572=1213.000,80.773,-47.460,-178.799,5.667,148.640
C03573=1212.995,81.041,-47.479,-178.796,5.669,148.639
C03574=1212.990,81.310,-47.498,-178.794,5.669,148.639
C03575=1212.985,81.578,-47.517,-178.791,5.670,148.638
C03576=1212.979,81.847,-47.536,-178.788,5.671,148.637
C03577=1212.974,82.096,-47.554,-178.786,5.672,148.637
C03578=1212.969,82.346,-47.572,-178.783,5.673,148.636
C03579=1212.965,82.595,-47.590,-178.780,5.673,148.636
C03580=1212.960,82.844,-47.608,-178.778,5.674,148.635
C03581=1212.954,83.094,-47.625,-178.775,5.676,148.635
C03582=1212.949,83.343,-47.643,-178.772,5.676,148.634
C03583=1212.945,83.592,-47.661,-178.770,5.677,148.634
C03584=1212.940,83.841,-47.679,-178.768,5.678,148.633
C03585=1212.935,84.090,-47.697,-178.765,5.678,148.632
C03586=1212.930,84.340,-47.715,-178.762,5.680,148.632
C03587=1212.925,84.589,-47.732,-178.760,5.681,148.631
C03588=1212.920,84.839,-47.751,-178.757,5.681,148.630
C03589=1212.915,85.088,-47.769,-178.755,5.682,148.630
C03590=1212.910,85.338,-47.787,-178.752,5.683,148.629
C03591=1212.906,85.587,-47.805,-178.749,5.684,148.629
C03592=1212.901,85.836,-47.823,-178.747,5.685,148.628
C03593=1212.896,86.085,-47.840,-178.744,5.686,148.628
C03594=1212.891,86.334,-47.858,-178.742,5.686,148.627
C03595=1212.886,86.583,-47.876,-178.740,5.687,148.627
C03596=1212.881,86.833,-47.894,-178.736,5.689,148.626
C03597=1212.877,87.083,-47.913,-178.734,5.689,148.625
C03598=1212.872,87.332,-47.931,-178.732,5.690,148.625
C03599=1212.867,87.581,-47.949,-178.729,5.691,148.624
C03600=1212.862,87.830,-47.967,-178.726,5.692,148.624
C03601=1212.857,88.079,-47.985,-178.724,5.693,148.623
C03602=1212.852,88.328,-48.003,-178.721,5.694,148.623
C03603=1212.847,88.578,-48.021,-178.718,5.694,148.622
C03604=1212.843,88.827,-48.039,-178.716,5.695,148.621
C03605=1212.838,89.077,-48.057,-178.713,5.696,148.621
C03606=1212.833,89.326,-48.075,-178.711,5.697,148.620
C03607=1212.828,89.575,-48.093,-178.708,5.698,148.620
C03608=1212.823,89.824,-48.111,-178.706,5.699,148.619
C03609=1212.818,90.073,-48.129,-178.703,5.700,148.619
C03610=1212.814,90.323,-48.147,-178.700,5.701,148.618
C03611=1212.808,90.573,-48.166,-178.698,5.702,148.617
C03612=1212.803,90.822,-48.184,-178.696,5.702,148.617
C03613=1212.799,91.071,-48.202,-178.692,5.704,148.616
C03614=1212.794,91.320,-48.220,-178.690,5.704,148.616
C03615=1212.789,91.570,-48.238,-178.688,5.705,148.615
C03616=1212.784,91.819,-48.256,-178.685,5.706,148.615
C03617=1212.780,92.068,-48.275,-178.682,5.708,148.614
C03618=1212.775,92.317,-48.293,-178.680,5.708,148.614
C03619=1212.769,92.567,-48.311,-178.677,5.709,148.613
C03620=1212.765,92.816,-48.330,-178.675,5.710,148.612
C03621=1212.760,93.066,-48.348,-178.672,5.711,148.612
C03622=1212.755,93.315,-48.366,-178.669,5.712,148.611
C03623=1212.751,93.563,-48.384,-178.667,5.713,148.611
C03624=1212.745,93.813,-48.403,-178.664,5.713,148.610
C03625=1212.741,94.063,-48.421,-178.662,5.715,148.610
C03626=1212.736,94.312,-48.439,-178.659,5.716,148.609
C03627=1212.731,94.561,-48.457,-178.657,5.716,148.608
C03628=1212.727,94.810,-48.476,-178.654,5.717,148.608
C03629=1212.721,95.060,-48.495,-178.651,5.719,148.607
C03630=1212.716,95.309,-48.513,-178.649,5.720,148.607
C03631=1212.711,95.558,-48.531,-178.646,5.720,148.606
C03632=1212.707,95.807,-48.550,-178.644,5.721,148.606
C03633=1212.702,96.057,-48.568,-178.641,5.723,148.605
C03634=1212.697,96.306,-48.586,-178.639,5.723,148.605
C03635=1212.693,96.555,-48.606,-178.636,5.724,148.604
C03636=1212.688,96.804,-48.623,-178.634,5.725,148.603
C03637=1212.682,97.054,-48.642,-178.631,5.726,148.603
C03638=1212.678,97.302,-48.661,-178.628,5.727,148.602
C03639=1212.673,97.552,-48.679,-178.626,5.728,148.602
C03640=1212.668,97.802,-48.697,-178.623,5.729,148.601
C03641=1212.663,98.050,-48.716,-178.621,5.730,148.601
C03642=1212.659,98.300,-48.735,-178.618,5.731,148.600
C03643=1212.654,98.549,-48.753,-178.616,5.731,148.600
C03644=1212.648,98.798,-48.772,-178.613,5.733,148.599
C03645=1212.644,99.048,-48.790,-178.610,5.733,148.598
C03646=1212.639,99.297,-48.809,-178.608,5.734,148.598
C03647=1212.634,99.546,-48.828,-178.605,5.736,148.597
C03648=1212.630,99.796,-48.846,-178.603,5.737,148.597
C03649=1212.625,100.045,-48.865,-178.600,5.737,148.596
C03650=1212.619,100.294,-48.883,-178.598,5.738,148.596
C03651=1212.615,100.543,-48.902,-178.595,5.740,148.595
C03652=1212.610,100.793,-48.920,-178.592,5.740,148.595
C03653=1212.605,101.041,-48.940,-178.590,5.741,148.594
